(* POU TCP_Logger/LogEv, ST *)
FUNCTION LogEv : BOOL
VAR_INPUT
	Level	: en_Logger_ErrLev;
	Object  : en_SYS_Objects;
	Index	: WORD;
	Error	: WORD;
	Message : STRING;
END_VAR
VAR
	s1 : STRING(160);
	i  : INT;
END_VAR
(* Execute error level operations *)
CASE Level OF
	EL_Wrn: 		Sys.Warning:=TRUE;
	EL_Alarm: 		Sys.Alarm  :=TRUE;
	EL_AlarmStop: 	Sys.Alarm  :=TRUE; (* GO TO STOP STATE!! *)
END_CASE

(* Fill lastlog list *)
s1:=CONCAT(Sys.Time_LogString,';Lev=');
s1:=CONCAT(s1,INT_TO_STRING(Level));
s1:=CONCAT(s1,';Obj=');
s1:=CONCAT(s1,INT_TO_STRING(Object));
s1:=CONCAT(s1,';Idx=');
s1:=CONCAT(s1,WORD_TO_STRING(Index));
s1:=CONCAT(s1,';Err=');
s1:=CONCAT(s1,WORD_TO_STRING(Error));
Sys.LastLogs_Dat[Sys.LastLogs_Idx]:=s1;
Sys.LastLogs_Msg[Sys.LastLogs_Idx]:=Message;
Sys.LastLogs_Idx:=Sys.LastLogs_Idx+1;
IF Sys.LastLogs_Idx>5 THEN Sys.LastLogs_Idx:=0; END_IF

(*---------------------------------------------------------------*)
	Logger_Head();
(*---------------------------------------------------------------*)

(* Insert ERR *)
s1:=CONCAT('&ERR=',INT_TO_STRING(Level));
s1:=CONCAT(s1,';');
s1:=CONCAT(s1,INT_TO_STRING(Object));
s1:=CONCAT(s1,';');
s1:=CONCAT(s1,WORD_TO_STRING(Index));
s1:=CONCAT(s1,';');
s1:=CONCAT(s1,WORD_TO_STRING(Error));
s1:=CONCAT(s1,';');
ADDSTRING(ADR(Logger.TData), ADR(s1), Logger.TLen);
s1:=Message;
STR_NOSPACES(ADR(s1));
ADDSTRING(ADR(Logger.TData), ADR(s1), Logger.TLen);

(*---------------------------------------------------------------*)
	Logger_Send();
(*---------------------------------------------------------------*)
END_FUNCTION

(* POU Utils Functions/STR_NOSPACES, ST *)
FUNCTION STR_NOSPACES : BOOL (* Replace spaces and bad chars with allowed ones, used as HTTP-GET validator *)
VAR_INPUT
	pString: POINTER TO BYTE;
END_VAR
VAR
END_VAR
WHILE pString^<>0 DO
	IF pString^=16#20 (* space *) THEN pString^:=16#5F; (*'_'*) END_IF
	pString:=pString+1;
END_WHILE
END_FUNCTION

(* POU Utils Functions/AVERAGE_DINT, ST *)
FUNCTION_BLOCK AVERAGE_DINT
VAR_INPUT
	IN: 	DINT;
END_VAR
VAR_OUTPUT
	HI:		DINT;
	AVG:	DINT;
	LOW:	DINT;
	ERR:	BOOL;
END_VAR
VAR
	sum:	REAL;
	cnt:	WORD;
END_VAR
IF cnt>=65000 THEN
	ERR:=TRUE;
	Read();
	sum := sum - DINT_TO_REAL(AVG);
	cnt := cnt - 1;
END_IF

sum := sum + DINT_TO_REAL(IN);
cnt := cnt + 1;

IF IN<LOW THEN LOW:=IN; END_IF
IF IN>HI  THEN HI :=IN; END_IF
END_FUNCTION_BLOCK
ACTION Read:
AVG := REAL_TO_DINT(sum/cnt);
END_ACTION
ACTION Reset:
HI:=IN;
AVG:=IN;
LOW:=IN;
ERR:=FALSE;

sum:=DINT_TO_REAL(IN);
cnt:=1;
END_ACTION

(* POU Utils Functions/AVERAGE_INT, ST *)
FUNCTION_BLOCK AVERAGE_INT
VAR_INPUT
	IN: 	INT;
END_VAR
VAR_OUTPUT
	HI:		INT;
	AVG:	INT;
	LOW:	INT;
	ERR:	BOOL;
END_VAR
VAR
	sum:	DINT;
	cnt:	WORD;
END_VAR
IF cnt>=65000 THEN
	ERR:=TRUE;
	Read();
	sum := sum - AVG;
	cnt := cnt - 1;
END_IF

sum := sum + IN;
cnt := cnt + 1;

IF IN<LOW THEN LOW:=IN; END_IF
IF IN>HI  THEN HI :=IN; END_IF
END_FUNCTION_BLOCK
ACTION Read:
AVG := DINT_TO_INT(sum/cnt);
END_ACTION
ACTION Reset:
HI:=IN;
AVG:=IN;
LOW:=IN;
ERR:=FALSE;

sum:=IN;
cnt:=1;
END_ACTION

(* POU Utils Functions/AVERAGE_T, ST *)
FUNCTION_BLOCK AVERAGE_T
VAR_INPUT
	IN: 	INT;
END_VAR
VAR_OUTPUT
	HI:		INT;
	AVG:	INT;
	LOW:	INT;
	ERR:	BOOL;
END_VAR
VAR
	sum:	DINT;
	cnt:	WORD;
END_VAR
IF cnt>=65000 THEN
	ERR:=TRUE;
	Read();
	sum := sum - AVG;
	cnt := cnt + 1;
END_IF

sum := sum + IN;
cnt := cnt + 1;

IF IN<LOW THEN  LOW:=IN; END_IF
IF IN>HI  THEN HI :=IN; END_IF
END_FUNCTION_BLOCK
ACTION Read:
AVG := DINT_TO_INT(sum/cnt);
END_ACTION
ACTION Reset:
HI:=IN;
AVG:=IN;
LOW:=IN;
ERR:=FALSE;

sum:=IN;
cnt:=1;
END_ACTION

(* POU Utils Functions/BUILD_16TO32, ST *)
FUNCTION BUILD_16TO32 : DWORD
VAR_INPUT
		pSource	:	POINTER TO WORD;
END_VAR
VAR
		Data	:	DWORD;
END_VAR
Data := WORD_TO_DWORD(pSource^);
pSource := pSource + 1;
Data := Data + WORD_TO_DWORD(pSource^) * 65536;

BUILD_16TO32 := Data;
END_FUNCTION

(* POU Utils Functions/COPY_32SWAP16, ST *)
FUNCTION COPY_32SWAP16:BOOL
VAR_INPUT
	pSourceAddress		:POINTER TO ARRAY[1..2] OF WORD;
	pDestinationAddress	:POINTER TO ARRAY[1..2] OF WORD;
END_VAR
VAR
END_VAR
pDestinationAddress^[1]:=pSourceAddress^[2];
pDestinationAddress^[2]:=pSourceAddress^[1];
END_FUNCTION

(* POU Utils Functions/FLT_EVENT, ST *)
FUNCTION_BLOCK FLT_EVENT
VAR_INPUT
	IN		: BOOL;
	INITEV	: BOOL:=TRUE;
END_VAR
VAR_OUTPUT
	EVH		: BOOL;
	EVL		: BOOL;
END_VAR
VAR
	init	: BOOL:=FALSE;
	old		: BOOL;
END_VAR
EVH:=FALSE;
EVL:=FALSE;

IF NOT init THEN
	init:=TRUE;
	IF INITEV THEN
		old := NOT IN;
	ELSE
		old := IN;
	END_IF
END_IF

IF old<>IN THEN
	old:=IN;
	IF IN THEN EVH:=TRUE; ELSE EVL:=TRUE; END_IF
END_IF
END_FUNCTION_BLOCK

(* POU Utils Functions/FLT_TIME, ST *)
FUNCTION_BLOCK FLT_TIME
VAR_INPUT
	IN		: BOOL;
	TTAP	: TIME:=T#5s;
	INITEV	: BOOL:=TRUE;
END_VAR
VAR_OUTPUT
	OUT		: BOOL;
	EVH		: BOOL;
	EVL		: BOOL;
END_VAR
VAR
	init	: BOOL:=FALSE;
	timer	: TON;
END_VAR
EVH:=FALSE;
EVL:=FALSE;

IF NOT init THEN
	init := TRUE;
	IF INITEV THEN
		OUT  := NOT IN;
	ELSE
		OUT  := IN;
	END_IF
END_IF

IF OUT<>IN THEN
	timer(IN:=TRUE,PT:=TTAP);
	IF timer.Q THEN
		OUT:=IN;
		timer(IN:=FALSE);
		IF OUT THEN EVH:=TRUE; ELSE EVL:=TRUE; END_IF
	END_IF
ELSE
	timer(IN:=FALSE);
END_IF
END_FUNCTION_BLOCK

(* POU Utils Functions/LAMP_AL_GENERALE, ST *)
FUNCTION_BLOCK LAMP_AL_GENERALE
VAR_INPUT

	Allarme: BOOL;
	Warning: BOOL;
END_VAR
VAR_OUTPUT
	SistemaOK:BOOL;
	SistemaInAllarme:BOOL;
	SistemaWarning:BOOL;
	AllarmeLampada:BOOL;
END_VAR
VAR
	Lampeggio:BLINK;
END_VAR
IF Allarme THEN       					(* Se Allarme Attivo Lucde fissa ON *)
	SistemaInAllarme:=TRUE;
	SistemaWarning:=FALSE;
	AllarmeLampada:=TRUE;
ELSIF Warning THEN					(* Se Allarme Attivo Lucde fissa pulse *)
	SistemaInAllarme:=FALSE;
	SistemaWarning:=TRUE;
	Lampeggio(ENABLE:=TRUE , TIMELOW:=t#1s , TIMEHIGH:=t#1s , OUT=>AllarmeLampada );
ELSE
	SistemaInAllarme:=FALSE;
	SistemaWarning:=FALSE;
	AllarmeLampada:=FALSE;
END_IF
END_FUNCTION_BLOCK

(* POU Utils Functions/LINEAR, ST *)
FUNCTION LINEAR : REAL (* Linear interpolation *)
VAR_INPUT
	X_In	: REAL;
	P1_X	: REAL;
	P1_Y	: REAL;
	P2_X	: REAL;
	P2_Y	: REAL;
END_VAR
VAR
END_VAR
LINEAR:=P1_Y+(((P2_Y-P1_Y)*(X_In-P1_X))/(P2_X-P1_X));
END_FUNCTION

(* POU Utils Functions/LINEAR_BAD, ST *)
FUNCTION LINEAR_BAD : INT (* Linear interpolation *)
VAR_INPUT
	PuntoMinX	: INT;
	PuntoMaxX	: INT;
	ValIn		: INT;
	PuntoMinY	: REAL;
	PuntoMaxY	: REAL;
	Decimali	: BYTE;
END_VAR
VAR
	Gain				: REAL;
	PuntoMinX_R			: REAL;
	PuntoMaxX_R			: REAL;
	Linearizzazione_R	: REAL;
END_VAR
PuntoMinX_R:=INT_TO_REAL(PuntoMinX);
PuntoMaxX_R:=INT_TO_REAL(PuntoMaxX);

Gain:=(PuntoMaxX_R-PuntoMinX_R)/(PuntoMaxY-PuntoMinY);	(* Calcolo in guadagno per la linarizzazione *)
Linearizzazione_R:=PuntoMinx+(Gain*(ValIn-PuntoMinY));	(* Ottengo il valore linearizzato *)

LINEAR_BAD:=REAL_TO_INT(Linearizzazione_R*(EXPT(10, Decimali)));  (* Ottengo intero con i decimai voluti *)
END_FUNCTION

(* POU Utils Functions/MEAN_T, ST *)
FUNCTION MEAN_T : INT
VAR_INPUT
		T1		:	INT;
		T2		:	INT;

		THR_L	:	INT;
		THR_H	:	INT;
END_VAR
VAR
		Tmean	:	INT;
END_VAR
IF T1 >= THR_L AND T1 <= THR_H THEN

	IF T2 >= THR_L AND T2 <= THR_H THEN
		Tmean := (T1 + T2)/2;
	ELSE
		Tmean := T1;
	END_IF
ELSE
	IF T2 >= THR_L AND T2 <= THR_H THEN
		Tmean := T2;
	ELSE
		Tmean := 16#7FFF;	(* No valid temperature data has been passed *)
	END_IF
END_IF

MEAN_T := Tmean;
END_FUNCTION

(* POU Utils Functions/MEMCLR, ST *)
FUNCTION MEMCLR:BOOL
VAR_INPUT
	pDestinationAddress:POINTER TO ARRAY[1..2] OF BYTE;
	BytesToClear:WORD;
END_VAR
VAR
END_VAR
WHILE (BytesToClear > 0) DO
	pDestinationAddress^[1]:=0;
	pDestinationAddress:=ADR(pDestinationAddress^[2]); (* increment destination *)
	BytesToClear:=BytesToClear -1; (* decrement number of bytes to copy *)
END_WHILE
END_FUNCTION

(* POU Utils Functions/MUX_T, ST *)
FUNCTION MUX_T : INT
(* Manage temperatures measured by different probes in the same room/environment, considering possible probe measurement errors *)
VAR_INPUT
	T1		:	INT;
	T2		:	INT;
	T3		:	INT;
	(*T4		:	INT := 0;*)

	Err1	:	BOOL := TRUE;
	Err2	:	BOOL := TRUE;
	Err3	:	BOOL := TRUE;
	(*Err4	:	BOOL := TRUE;*)

	Used	:	BYTE;

END_VAR
VAR
	Sum		:	INT;
	count	:	BYTE;
END_VAR
CASE Used OF

	1:	(* T1 passed *)
		IF Err1 THEN
			Sum := 16#7FFF;
		ELSE
			Sum := T1;
			count := 1;
		END_IF

	2:	(* T1, T2 passed *)
		IF Err1 THEN
			IF Err2 THEN
				Sum := 16#7FFF;
			ELSE
				Sum := T2;
				count := 1;
			END_IF
		ELSE
			IF Err2 THEN
				Sum := T1;
				count := 1;
			ELSE
				Sum := T1 + T2;
				count := 2;
			END_IF
		END_IF

	3:	(* T1, T2, T3 passed *)
		IF Err1 THEN
			IF Err2 THEN
				IF Err3 THEN
					Sum := 16#7FFF;
				ELSE
					Sum := T3;
					count := 1;
				END_IF
			ELSE
				IF Err3 THEN
					Sum := T2;
					count := 1;
				ELSE
					Sum := T2 + T3;
					count := 2;
				END_IF
			END_IF
		ELSE
			IF Err2 THEN
				IF Err3 THEN
					Sum := T1;
					count := 1;
				ELSE
					Sum := T1 + T3;
					count := 2;
				END_IF
			ELSE
				IF Err3 THEN
					Sum := T1 + T2;
					count := 2;
				ELSE
					Sum := T1 + T2 + T3;
					count := 3;
				END_IF
			END_IF
		END_IF
(*
	4:
		IF Err1 THEN
			IF Err2 THEN
				IF Err3 THEN
					IF Err4 THEN
						Sum := 16#7FFF;
					ELSE
						Sum := T4;
						count := 1;
					END_IF
				ELSE
					IF Err4 THEN
						Sum := T3;
						count := 1;
					ELSE
						Sum := T3 + T4;
						count := 2;
					END_IF
				END_IF
			ELSE
				IF Err3 THEN
					IF Err4 THEN
						Sum := T2;
						count := 1;
					ELSE
						Sum := T2 + T4;
						count := 2;
					END_IF
				ELSE
					IF Err4 THEN
						Sum := T2 + T3;
						count := 2;
					ELSE
						Sum := T2 + T3 + T4;
						count := 3;
					END_IF
				END_IF
			END_IF
		ELSE
			IF Err2 THEN
				IF Err3 THEN
					IF Err4 THEN
						Sum := T1;
					ELSE
						Sum := T1 + T4;
						count := 2;
					END_IF
				ELSE
					IF Err4 THEN
						Sum := T1 + T3;
						count := 2;
					ELSE
						Sum := T1 + T3 + T4;
						count := 3;
					END_IF
				END_IF
			ELSE
				IF Err3 THEN
					IF Err4 THEN
						Sum := T1 + T2;
						count := 2;
					ELSE
						Sum := T1 + T2 + T4;
						count := 3;
					END_IF
				ELSE
					IF Err4 THEN
						Sum := T1 + T2 + T3;
						count := 3;
					ELSE
						Sum := T1 + T2 + T3 + T4;
						count := 4;
					END_IF
				END_IF
			END_IF
		END_IF
*)
END_CASE

IF Sum = 16#7FFF THEN
	(* No valid data -> return default *)
	MUX_T := Plant_DefaultTAmb;
ELSE
	(* Do average *)
	MUX_T := Sum/count;
END_IF
END_FUNCTION

(* POU Plant_Objects/obj_COOV_01, ST *)
FUNCTION_BLOCK obj_COOV_01
(* === ZIGBEE AMBIENT SENSORS MT-200 ===
   v1.0[07/05/05] - Create
*)
VAR CONSTANT
	LQI_Threshold		:	WORD := 10;		(* Zigbee link quality minimum value *)
	LowBattVoltage		:	WORD := 2700;		(* Battery is considered low when reaches 1.35V each *)
END_VAR
VAR_INPUT
	(* Settings *)
	ID				: BYTE;
	Address			: BYTE;

(*	Refresh_Period	: TIME:=t#5m;
	(* Controls *)
	Refresh_Auto	: BOOL:=TRUE; (* Enable automatic refresh *) *)
	(* Modbus *)
	Refresh_Now	:	BOOL;	(* Start immediately modbus state machine *)
	retryErrMax	:	BYTE := 2;


END_VAR
VAR_IN_OUT
	(* Interface *)
	ModBus		:obj_MODBUS;

END_VAR
VAR_OUTPUT
	(* Status *)
	Status_Log		: BYTE;
	Status_Vis 		: DWORD;
END_VAR
VAR


	state		:	INT;
	retry		:	BYTE;
	retryErr	:	BYTE;
	ReadTmr		:	TON := (PT:=T#5s);
	fModbusAlr:BOOL;


	AlarmCtr		: BYTE;
	WarningCtr		: BYTE;

	id_locale: BYTE;

	MB_RegistriLetti: ARRAY [0..20] OF INT;

	Quality			: FLT_EVENT;
	Battery			: FLT_EVENT;
	Alarm			: FLT_EVENT;

	ERR				: BOOL;
	fLQI			: BOOL;
	fBatt			: BOOL;
	StatusOK		: BYTE;			(* 0: Status OK, >=1: Alarm and/or warning		Incremented by 1 when Alarm or Wrn occurs,
									decremented by 1 when restored	*)

	TimeOutModBus: TON;
	ErroreComuModBus: BOOL;

	VerificaFuctionCode: INT;
	VerificaNodoLetto: INT;



END_VAR
(* stato creato per potere interrogare il nodo corretto *)
id_locale:=ID+6;

Stm();

checkAlarm();
END_FUNCTION_BLOCK
ACTION AddLogData:
Logger.s1:=INSERT('&COOV=',BYTE_TO_STRING(ID),5);
IF ID<10 THEN Logger.s1:=INSERT(Logger.s1,'0',5); END_IF


Logger.s1:=CONCAT(Logger.s1,INT_TO_STRING(MB_RegistriLetti[6]));	(* Misura del sensore CO2 – valore istantaneo  *)
Logger.s1:=CONCAT(Logger.s1,';');
Logger.s1:=CONCAT(Logger.s1,INT_TO_STRING(MB_RegistriLetti[4]));	(* Livello di Batteria (in millesimi di volt) *)
Logger.s1:=CONCAT(Logger.s1,';'); 
Logger.s1:=CONCAT(Logger.s1,WORD_TO_STRING(MB_RegistriLetti[3]));	(* Livello segnale radio dell'ultimo messaggio ricevuto dal dispositivo  *)
Logger.s1:=CONCAT(Logger.s1,';'); 

Logger.s1:=CONCAT(Logger.s1,BYTE_TO_STRING(Status_Log));
ADDSTRING(ADR(Logger.TData), ADR(Logger.s1), Logger.TLen);
END_ACTION
ACTION CheckAlarm:
(**** GEstione Log ad Evento *****)


(* (MB_RegistriLetti[3]) check Livello segnale radio dell'ultimo messaggio ricevuto dal dispositivo *)

IF (MB_RegistriLetti[3]) < LQI_Threshold THEN
	fLQI := FALSE;
	ERR := TRUE;
ELSE
	fLQI := TRUE;
	ERR := FALSE;
END_IF

Quality(IN:=fLQI);

IF Quality.EVL THEN
	LogEv(SEL((MB_RegistriLetti[3])<>0,EL_Alarm,EL_Wrn),EO_ZTHL,ID,SEL((MB_RegistriLetti[3])<>0,7,2),WORD_TO_STRING((MB_RegistriLetti[3])));
	Status_Log := SEL((MB_RegistriLetti[3])<>0,2,1);
	StatusOK := StatusOK + 1;
END_IF

IF Quality.EVH THEN StatusOK := SEL(StatusOK=0, StatusOK-1, 0); END_IF

(* If probe (node) is present proceed checking other warnings, otherwise don't transmit anything *)
IF (MB_RegistriLetti[3]) <> 0 THEN

	(* Check battery voltage *)

(* (MB_RegistriLetti[4]) check Livello di Batteria (in millesimi di volt) *)

	IF (MB_RegistriLetti[4]) < LowBattVoltage THEN fBatt := TRUE;
	ELSE fBatt := FALSE;
	END_IF


	Battery(IN:=fBatt);

	IF Battery.EVH  THEN
		LogEv(EL_Wrn,EO_ZTHL,ID,6,' ');
		StatusOK := StatusOK + 1;
	END_IF

	IF Battery.EVL THEN StatusOK := SEL(StatusOK=0, StatusOK-1, 0); END_IF

END_IF

Alarm(IN:=(StatusOK=0));

IF Alarm.EVH THEN
	Status_Log := 0;
	LogEv(EL_Log,EO_ZTHL,ID,1,'');
END_IF

IF Status_Log = 2 THEN Status_Vis := COLOR_RED;
ELSIF Status_Log = 1 THEN Status_Vis := COLOR_YELLOW;
ELSE Status_Vis := COLOR_GREEN;
END_IF
END_ACTION
ACTION Stm:
CASE state OF
	0:	(* Refresh time manager *)
		ReadTmr(IN:=NOT ReadTmr.Q);
		(*A tempo interrogo il nodo sempre che non ci sia qualcuno che lo sta interrogando in quel momento *)

		IF (ReadTmr.Q AND NodoDaInterrogareMB2=id_locale )OR Refresh_Now AND NOT InibiscoModbusMB2 THEN
			state := 10;
			ReadTmr.PT := T#5s;  (* moreno *)
			Refresh_Now := FALSE;
			InibiscoModbusMB2 := TRUE;
		END_IF

	(**** Leggo le Analogiche a Disposzione  ****)

	10:	(* richiedo lettura Holding Register   *)

		Modbus.MB_Query.SlaveAddress := Address;
		Modbus.MB_Query.FunctionCode := 4;
		ModBus.MB_Query.Read_StartAddress := 0 ;			(* richiedo lettura altri Parametri *)
		ModBus.MB_Query.Read_Quantity := 8;
		ModBus.MB_Start := TRUE;
		state := 20;

	20:	(* Risposta all'interrogazione *)
		IF NOT ModBus.MB_Start   THEN
			VerificaFuctionCode:=ModBus.MB_Resp.FunctionCode;
			VerificaNodoLetto:=ModBus.MB_Resp.SlaveAddress;

			IF ModBus.MB_MASTER.MB_Error<>0 THEN
				state := 300;
			ELSE

				MB_RegistriLetti[0] := ModBus.MB_Resp.Data[0];   	(* Vedi tabella *)
				MB_RegistriLetti[1] := ModBus.MB_Resp.Data[1];		(* Vedi tabella *)
				MB_RegistriLetti[2] := ModBus.MB_Resp.Data[2];		(* Vedi tabella *)
				MB_RegistriLetti[3] := ModBus.MB_Resp.Data[3];		(* Vedi tabella *)
				MB_RegistriLetti[4] := ModBus.MB_Resp.Data[4];		(* Vedi tabella *)
				MB_RegistriLetti[5] := ModBus.MB_Resp.Data[5];		(* Vedi tabella *)
				MB_RegistriLetti[6] := ModBus.MB_Resp.Data[6];		(* Vedi tabella *)
				MB_RegistriLetti[7] := ModBus.MB_Resp.Data[7];		(* Vedi tabella *)
				MB_RegistriLetti[8] := ModBus.MB_Resp.Data[8];		(* Vedi tabella *)
				MB_RegistriLetti[9] := ModBus.MB_Resp.Data[9];		(* Vedi tabella *)
				MB_RegistriLetti[10] := ModBus.MB_Resp.Data[10];		(* Vedi tabella *)
				MB_RegistriLetti[11] := ModBus.MB_Resp.Data[11];		(* Vedi tabella *)
				MB_RegistriLetti[12] := ModBus.MB_Resp.Data[12];		(* Vedi tabella *)
				MB_RegistriLetti[13] := ModBus.MB_Resp.Data[13];		(* Vedi tabella *)

				state := 295;
			END_IF
		END_IF


		295:
		IF NOT ModBus.MB_Start THEN
			IF ModBus.MB_MASTER.MB_Error<>0 THEN (*OR ModBus.MB_MASTER.MB_Error<>0 THEN*)
				state := 300;
			ELSE
				IF fModbusAlr THEN fModbusAlr := FALSE; END_IF
				NodoDaInterrogareMB2:=id_locale+1;
				InibiscoModbusMB2:=FALSE;
				retryErr := 0;
				retry := 0;
				state := 0;
					IF fModbusAlr=FALSE AND ErroreComuModBus=TRUE THEN
						LogEv(EL_Log,EO_CHI,ID,62,'ComunicazioneModBus_OK');
						ErroreComuModBus := FALSE;
				(*	WarningCtr := SEL(WarningCtr=0, WarningCtr-1, 0); *)
					END_IF


			END_IF
		END_IF



	(**** CHECK MODBUS ERROR ****)
	300: 	(* Release MODBUS *)
			InibiscoModbusMB2:=FALSE;
			(* Retries *)
			retry:=retry+1;
			IF retry>3 THEN
				retry:=0;

				(* Verify if slave is dead *)
				IF retryErr < retryErrMaX THEN
					retryErr := retryErr + 1;
				ELSE
					fModbusAlr := TRUE;
					(* Verify ModBus error	*)

					IF fModbusAlr AND ErroreComuModBus=FALSE THEN
						LogEv(EL_Alarm,EO_CHI,ID,61,CONCAT('ErroreModbus_',INT_TO_STRING(ModBus.MB_MASTER.MB_Error)));
						ErroreComuModBus := TRUE;
					END_IF
				END_IF

				END_IF
			Refresh_Now := FALSE;
			InibiscoModbusMB2:=FALSE;
			NodoDaInterrogareMB2:=id_locale+1;
			state:=0;
END_CASE




(* Controllo Time Out Ciclo ModBus *)

TimeOutModBus(In:=state<>0,PT:=t#30s);
IF TimeOutModBus.Q THEN
	State:=0;
	Refresh_Now:=TRUE;  (* Rilancio la lettura del nodo *)
	IF MODBUS.MB_Lock=TRUE THEN MODBUS.MB_Lock:=FALSE;END_IF
	IF InibiscoModbusMB2=TRUE THEN InibiscoModbusMB2:=FALSE;END_IF
END_IF
END_ACTION

(* POU Plant_Objects/obj_MODBUS, ST *)
FUNCTION_BLOCK obj_MODBUS
(* === MODBUS PROTOCOL INTERFACE ===
   v1.1[19/06/15] - Added new VARS allocation and searching
*)
VAR CONSTANT
	VARS_Max	: BYTE := 32;
END_VAR
VAR_INPUT
	(* Settings *)
	ID			: BYTE;
	COM			: BYTE;
	BAUDRATE	: COM_BAUDRATE;
	RS485		: BOOL := FALSE;

	N_STOPBits	:BYTE:=1;

	(* Interface *)
	MB_MASTER	: MODBUS_EXTENDED_MASTER;
	MB_Start	: BOOL;
	MB_Query	: typModbusExtendedQuery;
	MB_Resp		: typModbusResponse;
	MB_Lock		: BOOL;
	MB_timeOut	: TIME := t#500ms;

	(* Variables management *)
	VARS_En		: BOOL;
	VARS		: ARRAY [0..VARS_Max] OF typ_MODBUS_VAR;
	VARS_Check	: BOOL;
	VARS_Alarm	: BOOL;

	(* Variables allocation *)
	VAR_Pointer : POINTER TO ARRAY[0..99] OF WORD;
	VAR_Cfg		: POINTER TO typ_MODBUS_VAR;
END_VAR
VAR_OUTPUT
	(* Status *)
	Status_Log	: BYTE;
	Status_Vis	: DWORD;
END_VAR
VAR
	sta         : BYTE :=0;
	i			: BYTE;
	j			: BYTE;
	Alarm		: FLT_EVENT;
	
	VarTmr		: TON := (PT:=T#1s);
	VarSta		: BYTE; (* Status *)
	VarCnt		: BYTE; (* Scan counter *)
	VarRetry	: BYTE;
	VarAlarm	: BYTE; (* Last variable with errors *)
END_VAR
IF N_STOPBits=1 THEN MB_MASTER.csCOM_STOPBITS:=STOPBITS_1;END_IF
IF N_STOPBits=2 THEN MB_MASTER.csCOM_STOPBITS:=STOPBITS_2;END_IF

MB_MASTER(ENABLE:=TRUE,	ASCII_Mode:=FALSE, bCOM_PORT:=COM, cbCOM_BAUDRATE:=BAUDRATE, cpCOM_PARITY:=PARITY_NO,
		cbsCOM_BYTESIZE:=BS_8, cfCOM_FLOW_CONTROL:=SEL(RS485,NO_FLOW_CONTROL,HALFDUPLEX),
		tTIME_OUT:=MB_timeOut,	StartFunction:=MB_Start, ExtQuery:=MB_Query, Response:=MB_Resp);

(* Process variable management *)
IF VARS_En THEN VARS_Process(); END_IF

(* Check status *)
Alarm(IN:=(MB_MASTER.bInterfaceError<>0));
IF Alarm.EVH THEN
	LogEv(SEL(MB_MASTER.bInterfaceError<>3,EL_Wrn,EL_Alarm),EO_MODBUS,ID,1,BYTE_TO_STRING(MB_MASTER.bInterfaceError));
END_IF
IF Alarm.EVL THEN								(* Trigger a fall edge: MODBUS back working *)
	LogEv(EL_Log,EO_MODBUS,ID,2,'MODBUS_OK');
END_IF

(* Log/visu status *)
   IF Alarm.IN   THEN Status_Log:=2; Status_Vis:=COLOR_RED;
ELSIF Vars_Alarm THEN Status_Log:=1; Status_Vis:=COLOR_YELLOW;
  				 ELSE Status_Log:=0; Status_Vis:=COLOR_GREEN;
END_IF
END_FUNCTION_BLOCK
ACTION VAR_Search:
(* Search VAR with specific pointer if not found return first free VAR
	[Last VAR is not active... used as safe area...] 
*)
j:=VARS_Max;
FOR i := 0 TO VARS_Max-1 DO
	IF VARS[i].Variable=0 AND j>i THEN j:=i; END_IF
	IF VARS[i].Variable=VAR_Pointer THEN
		VAR_Cfg:=ADR(VARS[i]);
		RETURN;
	END_IF
END_FOR
VAR_Cfg:=ADR(VARS[j]);
END_ACTION
ACTION VARS_Process:
(* Update var timers *)
VarTmr(IN:=(NOT VarTmr.Q));
IF VarTmr.Q THEN
	FOR i := 0 TO VARS_Max DO
		IF VARS[i].Refresh_Cnt>0 THEN VARS[i].Refresh_Cnt:=VARS[i].Refresh_Cnt-1; END_IF
	END_FOR
	VARS_Check:=TRUE;
END_IF


(* Process status *)
CASE VarSta OF
	0: (* === Init *)
		VarCnt:=0;
		VarSta:=1;

	1: (* === Wait check signal *)
		IF VARS_Check THEN				(* Decremented "Refresh_Cnt" *)
			VARS_Check:=FALSE;
			VarCnt:=0;
			VarSta:=2;
		END_IF

	2: (* === Check loop *)
		IF NOT (MB_Lock OR MB_Start) THEN
			WHILE VarCnt<=(VARS_Max-1) AND VarSta=2 DO
				(* Check only active vars *)
				IF VARS[VarCnt].Variable<>0 THEN			(* "Variable" is a pointer to word, so if 0 no address *)
					(* Check var auto-refresh on timer checks *)
					IF VARS[VarCnt].Refresh_Time>0 AND VARS[VarCnt].Refresh_Cnt=0 THEN
						VARS[VarCnt].Refresh_Cnt:=VARS[VarCnt].Refresh_Time;
						VarSta:=3;
					END_IF
					(* Check refresh for change or request *)
					CASE VARS[VarCnt].FunCode OF
						5,6,15,16: (* Write functions *)
							IF VARS[VarCnt].Variable_Size=1 THEN
								IF VARS[VarCnt].Variable^<>VARS[VarCnt].Variable_Mirror THEN
									VARS[VarCnt].Variable_Mirror:=VARS[VarCnt].Variable^;
									VarSta:=3;
								END_IF
							ELSE
								IF VARS[VarCnt].Variable_Mirror<>0 THEN
									VARS[VarCnt].Variable_Mirror:=0;
									VarSta:=3;
								END_IF
							END_IF
						1,2,3,4: (* Read functions *)
							IF VARS[VarCnt].Variable_Mirror<>0 THEN
								VARS[VarCnt].Variable_Mirror:=0;
								VarSta:=3;
							END_IF
					END_CASE
				END_IF
				(* Process query *)
				IF VarSta=3 THEN
					MB_Lock:=TRUE;
					MB_Query.SlaveAddress:=VARS[VarCnt].SlaveAddress;
					MB_Query.FunctionCode:=VARS[VarCnt].FunCode;
					CASE VARS[VarCnt].FunCode OF
						16#5,16#6,16#F,16#10:
							MB_Query.Read_Quantity:=0;
							MB_Query.Read_StartAddress:=0;
							MB_Query.Write_StartAddress:=VARS[VarCnt].FunAddress;
							MB_Query.Write_Quantity:=VARS[VarCnt].Variable_Size;
							IF VARS[VarCnt].Variable_Size=200 THEN
								COPY_32SWAP16(VARS[VarCnt].Variable, ADR(MB_Query.Write_Data[0]));
							ELSIF VARS[VarCnt].Variable_Size>1 THEN
								MEMCPY(VARS[VarCnt].Variable, ADR(MB_Query.Write_Data[0]), 2*VARS[VarCnt].Variable_Size);
							ELSE
								MB_Query.Write_Data[0]:=VARS[VarCnt].Variable^;
							END_IF
						16#1,16#2,16#3,16#4:
							MB_Query.Read_StartAddress:=VARS[VarCnt].FunAddress;
							IF VARS[VarCnt].Variable_Size=200 THEN MB_Query.Read_Quantity:=2; ELSE
							  MB_Query.Read_Quantity:=VARS[VarCnt].Variable_Size;
							END_IF
							MB_Query.Write_StartAddress:=0;
							MB_Query.Write_Quantity:=0;
					END_CASE
					VarRetry:=0;
					MB_Start:=TRUE;
				ELSE
					VarCnt:=VarCnt+1;
				END_IF
			END_WHILE
			(* Check loop completed -> no actions *)
			IF VarSta=2 THEN VarSta:=1; END_IF
		END_IF

	3: (* === Wait & process MB response *)
		IF NOT MB_Start THEN
			IF MB_MASTER.MB_Error=0 THEN
				CASE VARS[VarCnt].FunCode OF
					1,2,3,4:
						IF VARS[VarCnt].Variable_Size=200 THEN
							COPY_32SWAP16(ADR(MB_Resp.Data), VARS[VarCnt].Variable);
						ELSIF VARS[VarCnt].Variable_Size>1 THEN
							MEMCPY(ADR(MB_Resp.Data), VARS[VarCnt].Variable, 2*VARS[VarCnt].Variable_Size);
						ELSE
							VARS[VarCnt].Variable^:=MB_Resp.Data[0];
						END_IF
				END_CASE
				MB_Lock:=FALSE;
				(* Signal error recovery *)
				IF VARS_Alarm=TRUE AND VarCnt=VarAlarm THEN
					LogEv(EL_Wrn,EO_MODBUS,ID,5,'');
					VARS_Alarm:=FALSE;
				END_IF
				(* Next var *)
				VarCnt:=VarCnt+1;
				VarSta:=2;
			ELSE
				IF VarRetry<3 THEN
					VarRetry:=VarRetry+1;
					MB_Start:=TRUE;
				ELSE
					MB_Lock:=FALSE;
					(* Signal error *)
					IF VARS_Alarm=FALSE THEN
						LogEv(EL_Wrn,EO_MODBUS,ID,3,INT_TO_STRING(MB_MASTER.MB_Error));
						VARS_Alarm:=TRUE;
						VarAlarm:=VarCnt-1;
					END_IF
					(* Next var *)
					VarCnt:=VarCnt+1;
					VarSta:=2;
				END_IF
			END_IF
		END_IF

ELSE
	VarSta:=0;
END_CASE
END_ACTION

(* POU Plant_Objects/obj_CRON, ST *)
FUNCTION_BLOCK obj_CRON
(* === CRONOGRAFO STANDARD ===
   v1.0[16/04/15] - Versioning
   v1.1[19/05/15] - Removed DB creation from previous year
*)
VAR_INPUT
	(* Settings *)
	ID			: BYTE;		(* Index of instanced object *)

	InitOK		: BOOL;
	Alarm		: BOOL;
	Warning		: BOOL;

	Profile		: typ_Cron_Profile; 				(* Profilo attivo *)
	ProfileNr	: BYTE;								(* Indice profilo attivo *)
	CalendarIdx : WORD;								(* Indice calendario attivo *)
	Jolly		: ARRAY[0..9] OF typ_Cron_Jolly;	(* Jolly attivi *)

END_VAR
VAR_IN_OUT
END_VAR
VAR_OUTPUT
	SetPoint		: INT;
	(* Status *)
	Status_Log		: BYTE;
	Status_Vis 		: DWORD;
END_VAR
VAR
	Buf: 	ARRAY[0..512] OF BYTE; (* AVOID THIS!! *)
	hFile: 	DWORD;
	sFile: 	STRING;
	sFile2: STRING;

	i:		WORD;
	t1:		DWORD;
	t2:		BOOL;

END_VAR
(* Check initialization *)
IF NOT InitOK THEN Init(); END_IF

(* Chrono *)
IF CalendarIdx<>Sys.Time_CT_Day THEN DB_Load(); END_IF
SetPoint:=Profile.Setpoint[Sys.Time_CT_Quarter];

(* Check jolly *)
FOR i := 0 TO 9 DO
	IF ( DT_TO_DWORD(Jolly[i].Start)>0  AND Jolly[i].End>Jolly[i].Start AND
	     Jolly[i].Start<=Sys.Time_CT_DT AND Jolly[i].End>Sys.Time_CT_DT ) THEN
			SetPoint:=Jolly[i].Temp;
	END_IF
END_FOR


(* Status color *)
   IF Alarm   THEN Status_Log:=2; Status_Vis:=COLOR_RED;
ELSIF Warning THEN Status_Log:=1; Status_Vis:=COLOR_YELLOW;
              ELSE Status_Log:=0; Status_Vis:=COLOR_GREEN;
			  END_IF
END_FUNCTION_BLOCK
ACTION AddLogData:
Logger.s1:=INSERT('&CRON=',BYTE_TO_STRING(ID),5);
IF ID<10 THEN Logger.s1:=INSERT(Logger.s1,'0',5); END_IF

Logger.s1:=CONCAT(Logger.s1,INT_TO_STRING(SetPoint));			Logger.s1:=CONCAT(Logger.s1,';');

Logger.s1:=CONCAT(Logger.s1,WORD_TO_STRING(Status_Log));
ADDSTRING(ADR(Logger.TData), ADR(Logger.s1), Logger.TLen);
END_ACTION
ACTION DB_Create:
(* Create empty file *)
hFile:=SysFileOpen(FileName:=sFile, Mode:='w');

MEMCLR(pDestinationAddress:=ADR(Buf), BytesToClear:=SIZEOF(Buf));
FOR i := 0 TO 10239 BY 512 DO
	t1:=SysFileWrite(File:=hFile, Buffer:=ADR(Buf), Size:=512);		(* Clear created file (all bytes 0) *)
END_FOR
Buf[0]:=1;
t2:=SysFileSetPos(File:=hFile, Pos:=0);
t1:=SysFileWrite(File:=hFile, Buffer:=ADR(Buf), Size:=1);
SysFileClose(File:=hFile);
END_ACTION
ACTION DB_Load:
DB_SetName();

(* Open data file *)
hFile:=SysFileOpen(FileName:=sFile, Mode:='r');

(* File not found *)
IF hFile=0 THEN
	Warning:=TRUE;
	LogEv(EL_Wrn,EO_CRON,ID,1,'No_data_file');
	DB_Create();
	(* Reopen file *)
	hFile:=SysFileOpen(FileName:=sFile, Mode:='r');
	IF hfile=0 THEN
		Alarm:=TRUE;
		LogEv(EL_Alarm,EO_CRON,ID,3,'Filesystem_error');
		RETURN;
	END_IF
END_IF

(* Check version *)
SysFileRead(File:=hFile, Buffer:=ADR(Buf), Size:=1);
IF Buf[0]<>1 THEN
	IF NOT Alarm THEN
		Alarm:=TRUE;
		LogEv(EL_Alarm,EO_CRON,ID,2,'Bad_data_version');
	END_IF
	SysFileClose(File:=hFile);
	RETURN;
END_IF

(* Read Jolly data *)
t2:=SysFileSetPos(File:=hFile, Pos:=512);
t1:=SysFileRead(File:=hFile, Buffer:=ADR(Jolly), Size:=SIZEOF(Jolly));
(* Read active profile index *)
CalendarIdx:=Sys.Time_CT_Day;
t2:=SysFileSetPos(File:=hFile, Pos:=(1024+4*CalendarIdx));
t1:=SysFileRead(File:=hFile, Buffer:=ADR(ProfileNr), Size:=SIZEOF(ProfileNr));
(* Read active profile *)
t2:=SysFileSetPos(File:=hFile, Pos:=(3072+512*ProfileNr));
t1:=SysFileRead(File:=hFile, Buffer:=ADR(Profile), Size:=SIZEOF(Profile));

(* Close file and validate data *)
SysFileClose(File:=hFile);
END_ACTION
ACTION DB_SetName:
(* Create current filename 'yyyyCRnn.DAT' *)
sFile:=CONCAT(FilesPath,WORD_TO_STRING(Sys.Time_Year));
sFile:=CONCAT(STR1:=sFile, STR2:='CR');
IF ID<10 THEN
sFile:=CONCAT(STR1:=sFile, STR2:='0');
END_IF
sFile:=CONCAT(STR1:=sFile, STR2:=BYTE_TO_STRING(ID));
sFile:=CONCAT(STR1:=sFile, STR2:='.DAT');
END_ACTION
ACTION Init:
DB_Load();
InitOK:=TRUE;
END_ACTION

(* POU Plant_Objects/obj_CRON_EDITOR, ST *)
FUNCTION_BLOCK obj_CRON_EDITOR
(* === EDITOR CRONOGRAFO ===
   v1.0[16/04/15] - Versioning
   v1.1[19/05/15] - Create empty profile when not found
*)
VAR_INPUT

	(* Common selections *)
	CN_Sel:			BYTE:=1;
	CN_Act:			BYTE;
	CN_YSel:		WORD:=2015;
	CN_YAct:		WORD;

	(* Profile editor *)
	PR_Sel: 		BYTE:=1;
	PR_Act:			BYTE;
	PR_TT:			REAL;
	PR:				typ_Cron_Profile;
	(* Profile signals *)
	PR_Load:		BOOL;
	PR_Save:		BOOL;

	(* Calendar editor *)
	CA_Sel:			BYTE:=1; (* Calendar month selected *)
	CA_Act:			BYTE;    (* Calendar month active *)
	CA_DayF:		BYTE:=0;
	CA_DayL:		BYTE:=31;
	CA_TPR:			BYTE;
	CA:				typ_Cron_Calendar; (* Only used for first 32 entries *)
	(* Calendar signals *)
	CA_Load:		BOOL;
	CA_Save:		BOOL;

	(* Jolly editor *)
	JL:				ARRAY[0..9] OF typ_Cron_Jolly;
	(* Jolly signals *)
	JL_Load:		BOOL;
	JL_Save:		BOOL;

END_VAR
VAR_OUTPUT
	Message		: STRING;
END_VAR
VAR
	sFileName	: STRING;
	sFileMode	: STRING;
	hFile		: DWORD;
	Buf			: ARRAY[0..512] OF BYTE; (* AVOID THIS!! *)

	i			: WORD;
	ver			: BYTE;
	r1			: BOOL;
	r2			: DWORD;

END_VAR
IF PR_Load THEN PR_Load_Exe(); PR_Load:=FALSE; END_IF
IF PR_Save THEN PR_Save_Exe(); PR_Save:=FALSE; END_IF
IF CA_Load THEN CA_Load_Exe(); CA_Load:=FALSE; END_IF
IF CA_Save THEN CA_Save_Exe(); CA_Save:=FALSE; END_IF
IF JL_Load THEN JL_Load_Exe(); JL_Load:=FALSE; END_IF
IF JL_Save THEN JL_Save_Exe(); JL_Save:=FALSE; END_IF
END_FUNCTION_BLOCK
ACTION CA_Load_Exe:
sFileMode:='r';
FileOpen();

IF hFile<>0 THEN

	(* Read calendar month *)
	FOR i := 0 TO 31 DO
		r1:=SysFileSetPos(File:=hFile, Pos:=(1024 + ((CA_Sel-1)*32 + i)*4));
		r2:=SysFileRead(File:=hFile, Buffer:=ADR(CA.Profile[i]), Size:=1);
	END_FOR

	(* Close file *)
	SysFileClose(File:=hFile);

	(* Validate data *)
	CA_Act :=CA_Sel;
	CN_Act :=CN_Sel;
	CN_YAct:=CN_YSel;

	Message:='Calendar load OK';

END_IF
END_ACTION
ACTION CA_Save_Exe:
sFileMode:='a';
FileOpen();

IF hFile<>0 THEN

	(* Write calendar month *)
	FOR i := 0 TO 31 DO
		r1:=SysFileSetPos(File:=hFile, Pos:=(1024 + ((CA_Sel-1)*32 + i)*4));
		r2:=SysFileGetPos(hFile);
		r2:=SysFileWrite(File:=hFile, Buffer:=ADR(CA.Profile[i]), Size:=1);
	END_FOR

	(* Close file *)
	SysFileClose(File:=hFile);

	Message:='Calendar save OK';

END_IF
END_ACTION
ACTION FileOpen:
(* Create current filename 'yyyyCRnn.DAT' *)
sFileName:=CONCAT(FilesPath,WORD_TO_STRING(CN_YSel));
sFileName:=CONCAT(STR1:=sFileName, STR2:='CR');
IF CN_Sel<10 THEN
sFileName:=CONCAT(STR1:=sFileName, STR2:='0');
END_IF
sFileName:=CONCAT(STR1:=sFileName, STR2:=BYTE_TO_STRING(CN_Sel));
sFileName:=CONCAT(STR1:=sFileName, STR2:='.DAT');

(* Check file version and size! *)
(* ... *)

(* Open data file *)
hFile:=SysFileOpen(FileName:=sFileName, Mode:='r');

(* File not found *)
IF hFile=0 THEN
	Message:='File not found - created empty file';
	(* Create empty file *)
	hFile:=SysFileOpen(FileName:=sFileName, Mode:='w');
	MEMCLR(pDestinationAddress:=ADR(Buf), BytesToClear:=SIZEOF(Buf));
	FOR i := 0 TO 10239 BY 512 DO
		SysFileWrite(File:=hFile, Buffer:=ADR(Buf), Size:=512);
	END_FOR
	Buf[0]:=1;
	SysFileSetPos(File:=hFile, Pos:=0);
	SysFileWrite(File:=hFile, Buffer:=ADR(Buf), Size:=1);
END_IF

(* Close file *)
SysFileClose(File:=hFile);

(* Open data file *)
hFile:=SysFileOpen(FileName:=sFileName, Mode:=sFileMode);
END_ACTION
ACTION JL_Load_Exe:
sFileMode:='r';
FileOpen();

IF hFile<>0 THEN

	(* Read jolly *)
	r1:=SysFileSetPos(File:=hFile, Pos:=512);
	r2:=SysFileRead(File:=hFile, Buffer:=ADR(JL), Size:=SIZEOF(JL));

	(* Close file *)
	SysFileClose(File:=hFile);

	(* Validate data *)
	CN_Act:=CN_Sel;
	CN_YAct:=CN_YSel;

	Message:='Jolly load OK';

END_IF
END_ACTION
ACTION JL_Save_Exe:
sFileMode:='a';
FileOpen();

IF hFile<>0 THEN

	(* Write selected profile *)
	r1:=SysFileSetPos(File:=hFile, Pos:=512);
	r2:=SysFileWrite(File:=hFile, Buffer:=ADR(JL), Size:=SIZEOF(JL));

	(* Close file *)
	SysFileClose(File:=hFile);

	Message:='Jolly save OK';

END_IF
END_ACTION
ACTION PR_Load_Exe:
sFileMode:='r';
FileOpen();

IF hFile<>0 THEN

	(* Read selected profile *)
	r1:=SysFileSetPos(File:=hFile, Pos:=(3072 + 512*PR_Sel));
	r2:=SysFileRead(File:=hFile, Buffer:=ADR(PR), Size:=SIZEOF(PR));

	(* Close file *)
	SysFileClose(File:=hFile);

	(* Validate data *)
	PR_Act:=PR_Sel;
	CN_Act:=CN_Sel;
	CN_YAct:=CN_YSel;

	Message:='Profile load OK';

END_IF
END_ACTION
ACTION PR_Save_Exe:
sFileMode:='a';
FileOpen();

IF hFile<>0 THEN

	(* Write selected profile *)
	r1:=SysFileSetPos(File:=hFile, Pos:=(3072 + 512*PR_Sel));
	r2:=SysFileWrite(File:=hFile, Buffer:=ADR(PR), Size:=SIZEOF(PR));

	(* Close file *)
	SysFileClose(File:=hFile);

	Message:='Profile save OK';

END_IF
END_ACTION

(* POU Plant_Objects/obj_CRONTER, ST *)
FUNCTION_BLOCK obj_CRONTER
(* === THERMOSTAT ===
   v1.0[30/07/15] - Versioning
*)
VAR_INPUT
	(* Settings *)
	ID			: BYTE;		(* Index of instanced object *)

	InitOK		: BOOL;
	Alarm		: BOOL;
	Warning		: BOOL;

	Profile		: typ_Cron_Profile; 				(* Profilo attivo *)
	ProfileNr	: BYTE;								(* Indice profilo attivo *)
	CalendarIdx : WORD;								(* Indice calendario attivo *)
	Jolly		: ARRAY[0..9] OF typ_Cron_Jolly;	(* Jolly attivi *)

	Temperature	: INT;
	Local_MaxRunTAmb	:	INT;					(* Local maximum environment temperature, NOT "TAMB" *)

	Histeresys:INT; (* isteresi per la ripartenza del Comando ON*)
END_VAR
VAR_IN_OUT
END_VAR
VAR_OUTPUT
	SetPoint		: INT;
	Run				: BOOL;
	AntifreezeForce	: BOOL;
	RunCrono		: BOOL;

	(* Status *)
	Status_Log		: BYTE;
	Status_Vis 		: DWORD;
END_VAR
VAR
	Buf: 	ARRAY[0..512] OF BYTE; (* AVOID THIS!! *)
	hFile: 	DWORD;
	sFile: 	STRING;
	sFile2: STRING;

	i:		WORD;
	t1:		DWORD;
	t2:		BOOL;

END_VAR
(* Check initialization *)
IF NOT InitOK THEN Init(); END_IF

(* Check Temperature *)
(*IF Temperature < Local_MaxRunTAmb THEN*)

	(* LOCAL environment temperature lower than maximum allowed -> Proceed with SetPoint adjustment *)
	(* Chrono *)
	IF CalendarIdx<>Sys.Time_CT_Day THEN DB_Load(); END_IF
	SetPoint:=Profile.Setpoint[Sys.Time_CT_Quarter];

	(* Check jolly *)
	FOR i := 0 TO 9 DO
		IF ( DT_TO_DWORD(Jolly[i].Start)>0  AND Jolly[i].End>Jolly[i].Start AND
		     Jolly[i].Start<=Sys.Time_CT_DT AND Jolly[i].End>Sys.Time_CT_DT ) THEN
				SetPoint:=Jolly[i].Temp;
		END_IF
	END_FOR

(*
	IF SetPoint < 180 THEN
		(* Switch off the device *)
		Run := FALSE;
	ELSE
		(* Set according to feedback T - Histeresys of 1°C *)
		IF Temperature >= (SetPoint + 5) THEN
			Run := FALSE;
		ELSIF Temperature <= (SetPoint - 5) THEN
			Run := TRUE;
		END_IF

		(* Between "SetPoint-5" and "SetPoint+5" last state (ON or OFF) of "Run" is kept	*)
	END_IF
*)

(* Gestione uscita Crono *)
		IF SetPoint>0 THEN RunCrono := TRUE;
		ELSIF SetPoint=0 THEN RunCrono := FALSE;
		END_IF

(* GEstione uscita Cronotermostato *)


		IF Temperature >= (SetPoint) THEN
			Run := FALSE;
		ELSIF Temperature <= (SetPoint - Histeresys) THEN
			Run := TRUE;
		END_IF


(*ELSE
	(* Environment overtemperature: stop heating -> Stop device *)
	Run := FALSE;
END_IF
*)
(* Freeze warning: Switch on and heat! *)
(*IF Temperature < Plant_AntiFreezeTAmb THEN AntifreezeForce := TRUE;
ELSE AntifreezeForce := FALSE;
END_IF*)



(* Status color *)
   IF Alarm   THEN Status_Log:=2; Status_Vis:=COLOR_RED;
ELSIF Warning THEN Status_Log:=1; Status_Vis:=COLOR_YELLOW;
              ELSE Status_Log:=0; Status_Vis:=COLOR_GREEN;
			  END_IF
END_FUNCTION_BLOCK
ACTION AddLogData:
Logger.s1:=INSERT('&THER=',BYTE_TO_STRING(ID),5);
IF ID<10 THEN Logger.s1:=INSERT(Logger.s1,'0',5); END_IF

Logger.s1:=CONCAT(Logger.s1,INT_TO_STRING(SetPoint));			Logger.s1:=CONCAT(Logger.s1,';');

Logger.s1:=CONCAT(Logger.s1,WORD_TO_STRING(Status_Log));
ADDSTRING(ADR(Logger.TData), ADR(Logger.s1), Logger.TLen);
END_ACTION
ACTION DB_Create:
(* Create empty file *)
hFile:=SysFileOpen(FileName:=sFile, Mode:='w');

MEMCLR(pDestinationAddress:=ADR(Buf), BytesToClear:=SIZEOF(Buf));
FOR i := 0 TO 10239 BY 512 DO
	t1:=SysFileWrite(File:=hFile, Buffer:=ADR(Buf), Size:=512);		(* Clear created file (all bytes 0) *)
END_FOR
Buf[0]:=1;
t2:=SysFileSetPos(File:=hFile, Pos:=0);
t1:=SysFileWrite(File:=hFile, Buffer:=ADR(Buf), Size:=1);
SysFileClose(File:=hFile);
END_ACTION
ACTION DB_Load:
DB_SetName();

(* Open data file *)
hFile:=SysFileOpen(FileName:=sFile, Mode:='r');

(* File not found *)
IF hFile=0 THEN
	Warning:=TRUE;
	LogEv(EL_Wrn,EO_CRON,ID,1,'No_data_file');
	DB_Create();
	(* Reopen file *)
	hFile:=SysFileOpen(FileName:=sFile, Mode:='r');
	IF hfile=0 THEN
		Alarm:=TRUE;
		LogEv(EL_Alarm,EO_CRON,ID,3,'Filesystem_error');
		RETURN;
	END_IF
END_IF

(* Check version *)
SysFileRead(File:=hFile, Buffer:=ADR(Buf), Size:=1);
IF Buf[0]<>1 THEN
	IF NOT Alarm THEN
		Alarm:=TRUE;
		LogEv(EL_Alarm,EO_CRON,ID,2,'Bad_data_version');
	END_IF
	SysFileClose(File:=hFile);
	RETURN;
END_IF

(* Read Jolly data *)
t2:=SysFileSetPos(File:=hFile, Pos:=512);
t1:=SysFileRead(File:=hFile, Buffer:=ADR(Jolly), Size:=SIZEOF(Jolly));
(* Read active profile index *)
CalendarIdx:=Sys.Time_CT_Day;
t2:=SysFileSetPos(File:=hFile, Pos:=(1024+4*CalendarIdx));
t1:=SysFileRead(File:=hFile, Buffer:=ADR(ProfileNr), Size:=SIZEOF(ProfileNr));
(* Read active profile *)
t2:=SysFileSetPos(File:=hFile, Pos:=(3072+512*ProfileNr));
t1:=SysFileRead(File:=hFile, Buffer:=ADR(Profile), Size:=SIZEOF(Profile));

(* Close file and validate data *)
SysFileClose(File:=hFile);
END_ACTION
ACTION DB_SetName:
(* Create current filename 'yyyyCRnn.DAT' *)
sFile:=CONCAT(FilesPath,WORD_TO_STRING(Sys.Time_Year));
sFile:=CONCAT(STR1:=sFile, STR2:='CR');
IF ID<10 THEN
sFile:=CONCAT(STR1:=sFile, STR2:='0');
END_IF
sFile:=CONCAT(STR1:=sFile, STR2:=BYTE_TO_STRING(ID));
sFile:=CONCAT(STR1:=sFile, STR2:='.DAT');
END_ACTION
ACTION Init:
DB_Load();
InitOK:=TRUE;
END_ACTION

(* POU Plant_Objects/obj_GATEWAY_01, ST *)
FUNCTION_BLOCK obj_GATEWAY_01
(* === ZIGBEE AMBIENT SENSORS MT-200 ===
   v1.0[07/05/05] - Create
*)
VAR CONSTANT
	LQI_Threshold		:	WORD := 100;		(* Zigbee link quality minimum value *)
	LowBattVoltage		:	WORD := 270;		(* Battery is considered low when reaches 1.35V each *)
END_VAR
VAR_INPUT
	(* Settings *)
	ID				: BYTE;
	Address			: BYTE;

(*	Refresh_Period	: TIME:=t#5m;
	(* Controls *)
	Refresh_Auto	: BOOL:=TRUE; (* Enable automatic refresh *)*)

	(* Modbus *)
	Refresh_Now	:	BOOL;	(* Start immediately modbus state machine *)
	retryErrMax	:	BYTE := 2;

	(* Limits *)
	Tmin			: INT := 50;
	Tmax			: INT := 400;
END_VAR
VAR_IN_OUT
	(* Interface *)
	ModBus		:obj_MODBUS;

END_VAR
VAR_OUTPUT
	(* Status *)
	Status_Log		: BYTE;
	Status_Vis 		: DWORD;
END_VAR
VAR


	state		:	INT;
	retry		:	BYTE;
	retryErr	:	BYTE;
	ReadTmr		:	TON := (PT:=T#5s);
	fModbusAlr:BOOL;


	AlarmCtr		: BYTE;
	WarningCtr		: BYTE;

	id_locale: BYTE;

	MB_RegistriLetti: ARRAY [0..40] OF WORD;

	Quality			: FLT_EVENT;
	Battery			: FLT_EVENT;
	Temperature		: FLT_EVENT := (INITEV:=FALSE);
	Alarm			: FLT_EVENT;

	ERR				: BOOL;
	fLQI			: BOOL;
	fBatt			: BOOL;
	fTemp			: BOOL;

	StatusOK		: BYTE;			(* 0: Status OK, >=1: Alarm and/or warning		Incremented by 1 when Alarm or Wrn occurs,
																					decremented by 1 when restored	*)
	TimeOutModBus: TON;
	ErroreComuModBus: BOOL;

	VerificaFuctionCode: INT;
	VerificaNodoLetto: INT;


END_VAR
(* stato creato per potere interrogare il nodo corretto *)
id_locale:=ID + 12;

Stm();
END_FUNCTION_BLOCK
ACTION Stm:
CASE state OF
	0:	(* Refresh time manager *)
		ReadTmr(IN:=NOT ReadTmr.Q);
		(*A tempo interrogo il nodo sempre che non ci sia qualcuno che lo sta interrogando in quel momento *)

		IF (ReadTmr.Q AND NodoDaInterrogareMB2=id_locale )OR Refresh_Now AND NOT InibiscoModbusMB2 THEN
			state := 10;
			ReadTmr.PT := T#5s;  (* moreno *)
			Refresh_Now := FALSE;
			InibiscoModbusMB2 := TRUE;
		END_IF

	(**** Leggo le Analogiche a Disposzione  ****)

	10:	(* richiedo lettura Holding Register   *)

		Modbus.MB_Query.SlaveAddress := Address;
		Modbus.MB_Query.FunctionCode := 4;
		ModBus.MB_Query.Read_StartAddress := 0 ;			(* richiedo lettura altri Parametri *)
		ModBus.MB_Query.Read_Quantity := 20;
		ModBus.MB_Start := TRUE;
		state := 20;

	20:	(* Risposta all'interrogazione *)
		IF NOT ModBus.MB_Start   THEN
			VerificaFuctionCode:=ModBus.MB_Resp.FunctionCode;
			VerificaNodoLetto:=ModBus.MB_Resp.SlaveAddress;

			IF ModBus.MB_MASTER.MB_Error<>0 THEN
				state := 300;
			ELSE

				MB_RegistriLetti[0] := ModBus.MB_Resp.Data[0];   	(* Vedi tabella *)
				MB_RegistriLetti[1] := ModBus.MB_Resp.Data[1];		(* Vedi tabella *)
				MB_RegistriLetti[2] := ModBus.MB_Resp.Data[2];		(* Vedi tabella *)
				MB_RegistriLetti[3] := ModBus.MB_Resp.Data[3];		(* Vedi tabella *)
				MB_RegistriLetti[4] := ModBus.MB_Resp.Data[4];		(* Vedi tabella *)
				MB_RegistriLetti[5] := ModBus.MB_Resp.Data[5];		(* Vedi tabella *)
				MB_RegistriLetti[6] := ModBus.MB_Resp.Data[6];		(* Vedi tabella *)
				MB_RegistriLetti[7] := ModBus.MB_Resp.Data[7];		(* Vedi tabella *)
				MB_RegistriLetti[8] := ModBus.MB_Resp.Data[8];		(* Vedi tabella *)
				MB_RegistriLetti[9] := ModBus.MB_Resp.Data[9];		(* Vedi tabella *)
				MB_RegistriLetti[10] := ModBus.MB_Resp.Data[10];		(* Vedi tabella *)
				MB_RegistriLetti[11] := ModBus.MB_Resp.Data[11];		(* Vedi tabella *)
				MB_RegistriLetti[12] := ModBus.MB_Resp.Data[12];		(* Vedi tabella *)
				MB_RegistriLetti[13] := ModBus.MB_Resp.Data[13];		(* Vedi tabella *)
				MB_RegistriLetti[14] := ModBus.MB_Resp.Data[14];		(* Vedi tabella *)
				MB_RegistriLetti[15] := ModBus.MB_Resp.Data[15];		(* Vedi tabella *)
				MB_RegistriLetti[16] := ModBus.MB_Resp.Data[16];		(* Vedi tabella *)
				MB_RegistriLetti[17] := ModBus.MB_Resp.Data[17];		(* Vedi tabella *)
				MB_RegistriLetti[18] := ModBus.MB_Resp.Data[18];		(* Vedi tabella *)
				MB_RegistriLetti[19] := ModBus.MB_Resp.Data[19];		(* Vedi tabella *)

				Modbus.MB_Query.SlaveAddress := Address;
				Modbus.MB_Query.FunctionCode := 4;
				ModBus.MB_Query.Read_StartAddress := 20 ;			(* richiedo lettura altri Parametri *)
				ModBus.MB_Query.Read_Quantity := 19;
				ModBus.MB_Start := TRUE;
				state := 30;

			END_IF
		END_IF

	30:	(* Risposta all'interrogazione *)
		IF NOT ModBus.MB_Start   THEN
			VerificaFuctionCode:=ModBus.MB_Resp.FunctionCode;
			VerificaNodoLetto:=ModBus.MB_Resp.SlaveAddress;

			IF ModBus.MB_MASTER.MB_Error<>0 THEN
				state := 300;
			ELSE

				MB_RegistriLetti[20] := ModBus.MB_Resp.Data[0];   	(* Vedi tabella *)
				MB_RegistriLetti[21] := ModBus.MB_Resp.Data[1];		(* Vedi tabella *)
				MB_RegistriLetti[22] := ModBus.MB_Resp.Data[2];		(* Vedi tabella *)
				MB_RegistriLetti[23] := ModBus.MB_Resp.Data[3];		(* Vedi tabella *)
				MB_RegistriLetti[24] := ModBus.MB_Resp.Data[4];		(* Vedi tabella *)
				MB_RegistriLetti[25] := ModBus.MB_Resp.Data[5];		(* Vedi tabella *)
				MB_RegistriLetti[26] := ModBus.MB_Resp.Data[6];		(* Vedi tabella *)
				MB_RegistriLetti[27] := ModBus.MB_Resp.Data[7];		(* Vedi tabella *)
				MB_RegistriLetti[28] := ModBus.MB_Resp.Data[8];		(* Vedi tabella *)
				MB_RegistriLetti[29] := ModBus.MB_Resp.Data[9];		(* Vedi tabella *)
				MB_RegistriLetti[30] := ModBus.MB_Resp.Data[10];		(* Vedi tabella *)
				MB_RegistriLetti[31] := ModBus.MB_Resp.Data[11];		(* Vedi tabella *)
				MB_RegistriLetti[32] := ModBus.MB_Resp.Data[12];		(* Vedi tabella *)
				MB_RegistriLetti[33] := ModBus.MB_Resp.Data[13];		(* Vedi tabella *)
				MB_RegistriLetti[34] := ModBus.MB_Resp.Data[14];		(* Vedi tabella *)
				MB_RegistriLetti[35] := ModBus.MB_Resp.Data[15];		(* Vedi tabella *)
				MB_RegistriLetti[36] := ModBus.MB_Resp.Data[16];		(* Vedi tabella *)
				MB_RegistriLetti[37] := ModBus.MB_Resp.Data[17];		(* Vedi tabella *)
				MB_RegistriLetti[38] := ModBus.MB_Resp.Data[18];		(* Vedi tabella *)
				MB_RegistriLetti[39] := ModBus.MB_Resp.Data[19];		(* Vedi tabella *)

				state := 295;

			END_IF
		END_IF






		295:
		IF NOT ModBus.MB_Start THEN
			IF ModBus.MB_MASTER.MB_Error<>0 THEN (*OR ModBus.MB_MASTER.MB_Error<>0 THEN*)
				state := 300;
			ELSE
				IF fModbusAlr THEN fModbusAlr := FALSE; END_IF
				NodoDaInterrogareMB2:=id_locale+1;
				InibiscoModbusMB2:=FALSE;
				retryErr := 0;
				retry := 0;
				state := 0;
					IF fModbusAlr=FALSE AND ErroreComuModBus=TRUE THEN
						LogEv(EL_Log,EO_CHI,ID,62,'ComunicazioneModBus_OK');
						ErroreComuModBus := FALSE;
				(*	WarningCtr := SEL(WarningCtr=0, WarningCtr-1, 0); *)
					END_IF


			END_IF
		END_IF



	(**** CHECK MODBUS ERROR ****)
	300: 	(* Release MODBUS *)
			InibiscoModbusMB3:=FALSE;
			(* Retries *)
			retry:=retry+1;
			IF retry>3 THEN
				retry:=0;

				(* Verify if slave is dead *)
				IF retryErr < retryErrMaX THEN
					retryErr := retryErr + 1;
				ELSE
					fModbusAlr := TRUE;
					(* Verify ModBus error	*)

					IF fModbusAlr AND ErroreComuModBus=FALSE THEN
						LogEv(EL_Alarm,EO_CHI,ID,61,CONCAT('ErroreModbus_',INT_TO_STRING(ModBus.MB_MASTER.MB_Error)));
						ErroreComuModBus := TRUE;
					END_IF
				END_IF

			END_IF
			Refresh_Now := FALSE;
			InibiscoModbusMB2:=FALSE;
			NodoDaInterrogareMB2:=id_locale+1;
			state:=0;
END_CASE




(* Controllo Time Out Ciclo ModBus *)

TimeOutModBus(In:=state<>0,PT:=t#30s);
IF TimeOutModBus.Q THEN
	State:=0;
	Refresh_Now:=TRUE;  (* Rilancio la lettura del nodo *)
	IF MODBUS.MB_Lock=TRUE THEN MODBUS.MB_Lock:=FALSE;END_IF
	IF InibiscoModbusMB2=TRUE THEN InibiscoModbusMB2:=FALSE;END_IF
END_IF
END_ACTION

(* POU Plant_Objects/obj_MODBUS_ANZFRER_01, ST *)
FUNCTION_BLOCK obj_MODBUS_ANZFRER_01
VAR CONSTANT

	TimeOutModBus: TON;


END_VAR
VAR_INPUT
	ID			:	BYTE;
	Address		:	BYTE;
	(* Modbus *)
	Refresh_Now	:	BOOL;			(* Richiesta di lettura stato macchina Immediata  *)
	retryErrMax	:	BYTE := 2;

(*	IndirizzoDaScrivere: WORD;
	DatoDaScrivere: INT;
	ScriviDato: BOOL; *)

END_VAR
VAR_IN_OUT
	ModBus		:obj_MODBUS;

END_VAR
VAR_OUTPUT
	Status_Log	:	WORD;
	Status_Vis	:	DWORD;
END_VAR
VAR

	state		:	INT;
	retry		:	BYTE;
	retryErr	:	BYTE;
	ReadTmr		:	TON := (PT:=T#5s);
	fModbusAlr:BOOL;

(*	retry_write	:	BYTE;
	fWriteStatus:	BOOL;
	fWriteMode	:	BOOL;
	fWriteReset	:	BOOL; *)

	x: INT;

	VerificaFuctionCode: INT;
	VerificaNodoLetto: INT;
	ErroreComuModBus: BOOL;
	IndiceErrore: BYTE;

	MB_BitStato: ARRAY [0..450] OF BOOL;
	MB_RegistriLetti: ARRAY [0..450] OF INT;




	AddressRead: BYTE;
	index: BYTE;
	indexErr: BYTE;


	MB_V_L1_N: DWORD;
	MB_V_L2_N: DWORD;
	MB_V_L3_N: DWORD;
	MB_V_L1_L2: DWORD;
	MB_V_L1_L3: DWORD;
	MB_V_L2_L3: DWORD;
	MB_V_IL1: DWORD;
	MB_V_IL2: DWORD;
	MB_V_IL3: DWORD;
	MB_V_F: DWORD;
	MB_V_P: DWORD;
	MB_V_Q: DWORD;
	MB_V_P_F: DWORD;
	MB_IL1_MAX: DWORD;
	MB_IL2_MAX: DWORD;
	MB_IL3_MAX: DWORD;
	MB_PF_IL1: DWORD;
	MB_PF_IL2: DWORD;
	MB_PF_IL3: DWORD;
	MB_COSPI_IL1: DWORD;
	MB_COSPI_IL2: DWORD;
	MB_COSPI_IL3: DWORD;
	MB_V_P_AVG: DWORD;
	MB_V_P_MAX: DWORD;
	MB_V_Q_MAX: DWORD;
	MB_V_Q_AVG: DWORD;
	MB_V_KWh: DWORD;
	MB_V_kVAr: DWORD;
	MB_Rappenergia: DWORD;


	moreno: ARRAY [0..20] OF WORD;

END_VAR
(* Call ModBus state machine *)
Stm();


(* Seganalzione stato Frigorifero  *)
IF ErroreComuModBus OR MB_BitStato[6] OR MB_BitStato[7] THEN
		Status_Log:=2; Status_Vis:=16#2020F0;
(*	ELSIF Warning OR Warning2 THEN
		Status_Log:=1; Status_Vis:=16#20F0F0; *)
    ELSE
		Status_Log:=0;
		Status_Vis:=16#006000;
END_IF
END_FUNCTION_BLOCK
ACTION AddLogData:
Logger.s1:=INSERT('&ANZ=',BYTE_TO_STRING(ID),4);
IF ID<10 THEN Logger.s1:=INSERT(Logger.s1,'0',4); END_IF


	Logger.s1:=CONCAT(Logger.s1,(REAL_TO_STRING(DWORD_TO_REAL(MB_V_L1_N)/1000)));
	Logger.s1:=CONCAT(Logger.s1,';');
	Logger.s1:=CONCAT(Logger.s1,(REAL_TO_STRING(DWORD_TO_REAL(MB_V_L2_N)/1000)));
	Logger.s1:=CONCAT(Logger.s1,';');
	Logger.s1:=CONCAT(Logger.s1,(REAL_TO_STRING(DWORD_TO_REAL(MB_V_L3_N)/1000)));
	Logger.s1:=CONCAT(Logger.s1,';');
	Logger.s1:=CONCAT(Logger.s1,(REAL_TO_STRING(DWORD_TO_REAL(MB_V_L1_L2)/1000)));
	Logger.s1:=CONCAT(Logger.s1,';');
	Logger.s1:=CONCAT(Logger.s1,(REAL_TO_STRING(DWORD_TO_REAL(MB_V_L1_L3)/1000)));
	Logger.s1:=CONCAT(Logger.s1,';');
	Logger.s1:=CONCAT(Logger.s1,(REAL_TO_STRING(DWORD_TO_REAL(MB_V_L2_L3)/1000)));
	Logger.s1:=CONCAT(Logger.s1,';');

	Logger.s1:=CONCAT(Logger.s1,(REAL_TO_STRING(DWORD_TO_REAL(MB_V_F))));
	Logger.s1:=CONCAT(Logger.s1,';');

	Logger.s1:=CONCAT(Logger.s1,(REAL_TO_STRING(DWORD_TO_REAL(MB_V_IL1))));
	Logger.s1:=CONCAT(Logger.s1,';');
	Logger.s1:=CONCAT(Logger.s1,(REAL_TO_STRING(DWORD_TO_REAL(MB_V_IL2))));
	Logger.s1:=CONCAT(Logger.s1,';');
	Logger.s1:=CONCAT(Logger.s1,(REAL_TO_STRING(DWORD_TO_REAL(MB_V_IL3))));
	Logger.s1:=CONCAT(Logger.s1,';');

	Logger.s1:=CONCAT(Logger.s1,(REAL_TO_STRING(DWORD_TO_REAL(MB_IL1_MAX))));
	Logger.s1:=CONCAT(Logger.s1,';');
	Logger.s1:=CONCAT(Logger.s1,(REAL_TO_STRING(DWORD_TO_REAL(MB_IL1_MAX))));
	Logger.s1:=CONCAT(Logger.s1,';');
	Logger.s1:=CONCAT(Logger.s1,(REAL_TO_STRING(DWORD_TO_REAL(MB_IL1_MAX))));
	Logger.s1:=CONCAT(Logger.s1,';');


	Logger.s1:=CONCAT(Logger.s1,(REAL_TO_STRING(DWORD_TO_REAL(MB_PF_IL1))));
	Logger.s1:=CONCAT(Logger.s1,';');
	Logger.s1:=CONCAT(Logger.s1,(REAL_TO_STRING(DWORD_TO_REAL(MB_PF_IL2))));
	Logger.s1:=CONCAT(Logger.s1,';');
	Logger.s1:=CONCAT(Logger.s1,(REAL_TO_STRING(DWORD_TO_REAL(MB_PF_IL3))));
	Logger.s1:=CONCAT(Logger.s1,';');

	Logger.s1:=CONCAT(Logger.s1,(REAL_TO_STRING(DWORD_TO_REAL(MB_V_P))));
	Logger.s1:=CONCAT(Logger.s1,';');
	Logger.s1:=CONCAT(Logger.s1,(REAL_TO_STRING(DWORD_TO_REAL(MB_V_P_AVG))));
	Logger.s1:=CONCAT(Logger.s1,';');
	Logger.s1:=CONCAT(Logger.s1,(REAL_TO_STRING(DWORD_TO_REAL(MB_V_P_MAX))));
	Logger.s1:=CONCAT(Logger.s1,';');

	Logger.s1:=CONCAT(Logger.s1,(REAL_TO_STRING(DWORD_TO_REAL(MB_V_Q))));
	Logger.s1:=CONCAT(Logger.s1,';');
	Logger.s1:=CONCAT(Logger.s1,(REAL_TO_STRING(DWORD_TO_REAL(MB_V_Q_MAX))));
	Logger.s1:=CONCAT(Logger.s1,';');


	CASE MB_Rappenergia OF
		1:	Logger.s1:=CONCAT(Logger.s1,(REAL_TO_STRING(DWORD_TO_REAL(MB_V_KWh)/100)));
			Logger.s1:=CONCAT(Logger.s1,';');
			Logger.s1:=CONCAT(Logger.s1,(REAL_TO_STRING(DWORD_TO_REAL(MB_V_kVAr)/100)));
			Logger.s1:=CONCAT(Logger.s1,';');

		10:	Logger.s1:=CONCAT(Logger.s1,(REAL_TO_STRING(DWORD_TO_REAL(MB_V_KWh)/10)));
			Logger.s1:=CONCAT(Logger.s1,';');
			Logger.s1:=CONCAT(Logger.s1,(REAL_TO_STRING(DWORD_TO_REAL(MB_V_kVAr)/10)));
			Logger.s1:=CONCAT(Logger.s1,';');

		100:Logger.s1:=CONCAT(Logger.s1,(REAL_TO_STRING(DWORD_TO_REAL(MB_V_KWh))));
			Logger.s1:=CONCAT(Logger.s1,';');
			Logger.s1:=CONCAT(Logger.s1,(REAL_TO_STRING(DWORD_TO_REAL(MB_V_kVAr))));
			Logger.s1:=CONCAT(Logger.s1,';');

	END_CASE

	Logger.s1:=CONCAT(Logger.s1,WORD_TO_STRING(Status_Log));
	Logger.s1:=CONCAT(Logger.s1,';');

	Logger.s1:=CONCAT(Logger.s1,(REAL_TO_STRING(DWORD_TO_REAL(MB_COSPI_IL1))));
	Logger.s1:=CONCAT(Logger.s1,';');
	Logger.s1:=CONCAT(Logger.s1,(REAL_TO_STRING(DWORD_TO_REAL(MB_COSPI_IL2))));
	Logger.s1:=CONCAT(Logger.s1,';');
	Logger.s1:=CONCAT(Logger.s1,(REAL_TO_STRING(DWORD_TO_REAL(MB_COSPI_IL3))));
	Logger.s1:=CONCAT(Logger.s1,';');
	Logger.s1:=CONCAT(Logger.s1,'0');    (* 0=3-phase, 1 = mono phase *)


ADDSTRING(ADR(Logger.TData), ADR(Logger.s1), Logger.TLen);
END_ACTION
ACTION Stm:
CASE state OF
	0:	(* Refresh time manager *)
		ReadTmr(IN:=NOT ReadTmr.Q);
		(*A tempo interrogo il nodo sempre che non ci sia qualcuno che lo sta interrogando in quel momento *)

		IF (ReadTmr.Q AND NodoDaInterrogareANZ=Address )OR Refresh_Now AND NOT InibiscoModbusANZ THEN
			state := 10;
			ReadTmr.PT := T#5s;
			Refresh_Now := FALSE;
			InibiscoModbusANZ := TRUE;
		END_IF

	(**** Leggo le Analogiche a Disposzione  ****)

	10:	(* richiedo lettura Holding Registere Chiller  *)

		Modbus.MB_Query.SlaveAddress := Address;
		Modbus.MB_Query.FunctionCode := 3;
		ModBus.MB_Query.Read_StartAddress := 256 ;			(* richiedo lettura altri Parametri *)
		ModBus.MB_Query.Read_Quantity := 20;
		ModBus.MB_Start := TRUE;
		state := 20;

	20:	(* Risposta all'interrogazione *)
		IF NOT ModBus.MB_Start   THEN
			VerificaFuctionCode:=ModBus.MB_Resp.FunctionCode;
			VerificaNodoLetto:=ModBus.MB_Resp.SlaveAddress;

			IF ModBus.MB_MASTER.MB_Error<>0 THEN
				state := 300;
			ELSE
				MB_V_L1_N:= ModBus.MB_Resp.Data[0]*65536 +  ModBus.MB_Resp.Data[1];   	(* Vedi tabella *)
				MB_V_L2_N:= ModBus.MB_Resp.Data[2]*65536 +  ModBus.MB_Resp.Data[3];   	(* Vedi tabella *)
				MB_V_L3_N:= ModBus.MB_Resp.Data[4]*65536 +  ModBus.MB_Resp.Data[5];   	(* Vedi tabella *)
				MB_V_L1_L2:= ModBus.MB_Resp.Data[6]*65536 +  ModBus.MB_Resp.Data[7];   	(* Vedi tabella *)
				MB_V_L1_L3:= ModBus.MB_Resp.Data[8]*65536 +  ModBus.MB_Resp.Data[9];   	(* Vedi tabella *)
				MB_V_L2_L3:= ModBus.MB_Resp.Data[10]*65536 +  ModBus.MB_Resp.Data[11];   	(* Vedi tabella *)
				ModBus.MB_Query.Read_StartAddress := 268; 	(* richiedo lettura altri Parametri *)
				ModBus.MB_Query.Read_Quantity := 10;
				ModBus.MB_Start := TRUE;

				state := 30;
			END_IF
		END_IF

	30: (* Rispota Altri paramenti *)
		IF NOT ModBus.MB_Start  THEN

			IF ModBus.MB_MASTER.MB_Error<>0 THEN
				state := 300;
			ELSE
				MB_V_IL1:= ModBus.MB_Resp.Data[0]*65536 +  ModBus.MB_Resp.Data[1];   	(* Vedi tabella *)
				MB_V_IL2:= ModBus.MB_Resp.Data[2]*65536 +  ModBus.MB_Resp.Data[3];   	(* Vedi tabella *)
				MB_V_IL3:= ModBus.MB_Resp.Data[4]*65536 +  ModBus.MB_Resp.Data[5];   	(* Vedi tabella *)
				MB_V_F:= ModBus.MB_Resp.Data[6]*65536 +  ModBus.MB_Resp.Data[7];   	(* Vedi tabella *)
				MB_V_P:= ModBus.MB_Resp.Data[8]*65536 +  ModBus.MB_Resp.Data[9];   	(* Vedi tabella *)

				ModBus.MB_Query.Read_StartAddress := 278; (* richiedo lettura altri Parametri *)
				ModBus.MB_Query.Read_Quantity := 20;
				ModBus.MB_Start := TRUE;

				state := 40;
			END_IF
		END_IF



	40: (* Rispota Altri paramenti *)
		IF NOT ModBus.MB_Start  THEN

			IF ModBus.MB_MASTER.MB_Error<>0 THEN
				state := 300;
			ELSE
				MB_V_Q:= ModBus.MB_Resp.Data[0]*65536 +  ModBus.MB_Resp.Data[1];   	(* Vedi tabella *)
				MB_V_P_F:= ModBus.MB_Resp.Data[2]*65536 +  ModBus.MB_Resp.Data[3];   	(* Vedi tabella *)
				MB_V_KWh:= ModBus.MB_Resp.Data[4]*65536 +  ModBus.MB_Resp.Data[5];   	(* Vedi tabella *)
				MB_V_kVAr:= ModBus.MB_Resp.Data[6]*65536 +  ModBus.MB_Resp.Data[7];   	(* Vedi tabella *)
				MB_Rappenergia:= ModBus.MB_Resp.Data[8]*65536 +  ModBus.MB_Resp.Data[9];   	(* Vedi tabella *)

				ModBus.MB_Query.Read_StartAddress := 354; (* richiedo lettura altri Parametri *)
				ModBus.MB_Query.Read_Quantity := 20;
				ModBus.MB_Start := TRUE;

				state := 50;
			END_IF
		END_IF

	50: (* Rispota Altri paramenti *)
		IF NOT ModBus.MB_Start  THEN

			IF ModBus.MB_MASTER.MB_Error<>0 THEN
				state := 300;
			ELSE

				MB_V_P_AVG:= ModBus.MB_Resp.Data[0]*65536 +  ModBus.MB_Resp.Data[1];   	(* Vedi tabella *)
				MB_V_P_MAX:= ModBus.MB_Resp.Data[2]*65536 +  ModBus.MB_Resp.Data[3];   	(* Vedi tabella *)
				MB_IL1_MAX:= ModBus.MB_Resp.Data[4]*65536 +  ModBus.MB_Resp.Data[5];   	(* Vedi tabella *)
				MB_IL2_MAX:= ModBus.MB_Resp.Data[6]*65536 +  ModBus.MB_Resp.Data[7];   	(* Vedi tabella *)
				MB_IL3_MAX:= ModBus.MB_Resp.Data[8]*65536 +  ModBus.MB_Resp.Data[9];   	(* Vedi tabella *)

				ModBus.MB_Query.Read_StartAddress := 342; (* richiedo lettura altri Parametri *)
				ModBus.MB_Query.Read_Quantity := 20;
				ModBus.MB_Start := TRUE;

				state := 55;
			END_IF
		END_IF

	55: (* Rispota Altri paramenti *)
		IF NOT ModBus.MB_Start  THEN

			IF ModBus.MB_MASTER.MB_Error<>0 THEN
				state := 300;
			ELSE
				MB_PF_IL1:= ModBus.MB_Resp.Data[0]*65536 +  ModBus.MB_Resp.Data[1];   	(* Vedi tabella *)
				MB_PF_IL2:= ModBus.MB_Resp.Data[2]*65536 +  ModBus.MB_Resp.Data[3];   	(* Vedi tabella *)
				MB_PF_IL3:= ModBus.MB_Resp.Data[4]*65536 +  ModBus.MB_Resp.Data[5];   	(* Vedi tabella *)
				MB_COSPI_IL1:= ModBus.MB_Resp.Data[6]*65536 +  ModBus.MB_Resp.Data[7];   	(* Vedi tabella *)
				MB_COSPI_IL2:= ModBus.MB_Resp.Data[8]*65536 +  ModBus.MB_Resp.Data[9];   	(* Vedi tabella *)
				MB_COSPI_IL3:= ModBus.MB_Resp.Data[10]*65536 +  ModBus.MB_Resp.Data[11];   	(* Vedi tabella *)

				ModBus.MB_Query.Read_StartAddress := 422; (* richiedo lettura altri Parametri *)
				ModBus.MB_Query.Read_Quantity := 20;
				ModBus.MB_Start := TRUE;

				state := 60;
			END_IF
		END_IF

	60: (* Rispota Altri paramenti *)
		IF NOT ModBus.MB_Start  THEN

			IF ModBus.MB_MASTER.MB_Error<>0 THEN
				state := 300;
			ELSE
				MB_V_Q_MAX:= ModBus.MB_Resp.Data[0]*65536 +  ModBus.MB_Resp.Data[1];   	(* Vedi tabella *)
				MB_V_Q_AVG:= ModBus.MB_Resp.Data[2]*65536 +  ModBus.MB_Resp.Data[3];   	(* Vedi tabella *)

				(* ModBus.MB_Query.Read_StartAddress := 422; (* richiedo lettura altri Parametri *)
				ModBus.MB_Query.Read_Quantity := 20;
				ModBus.MB_Start := TRUE; *)

				state := 295;
			END_IF
		END_IF





		295:
		IF NOT ModBus.MB_Start THEN
			IF ModBus.MB_MASTER.MB_Error<>0 THEN (*OR ModBus.MB_MASTER.MB_Error<>0 THEN*)
				state := 300;
			ELSE
				IF fModbusAlr THEN fModbusAlr := FALSE; END_IF
				NodoDaInterrogareANZ:=Address+1;
				InibiscoModbusANZ:=FALSE;
				retryErr := 0;
				retry := 0;
				state := 0;
					IF fModbusAlr=FALSE AND ErroreComuModBus=TRUE THEN
						LogEv(EL_Log,EO_CHI,ID,62,'ComunicazioneModBus_OK');
						ErroreComuModBus := FALSE;
				(*	WarningCtr := SEL(WarningCtr=0, WarningCtr-1, 0); *)
					END_IF


			END_IF
		END_IF



	(**** CHECK MODBUS ERROR ****)
	300: 	(* Release MODBUS *)
			InibiscoModbusANZ:=FALSE;
			(* Retries *)
			retry:=retry+1;
			IF retry>3 THEN
				retry:=0;

				(* Verify if slave is dead *)
				IF retryErr < retryErrMaX THEN
					retryErr := retryErr + 1;
				ELSE
					fModbusAlr := TRUE;
					(* Verify ModBus error	*)

					IF fModbusAlr AND ErroreComuModBus=FALSE THEN
						LogEv(EL_Alarm,EO_CHI,ID,61,CONCAT('ErroreModbus_',INT_TO_STRING(ModBus.MB_MASTER.MB_Error)));
						ErroreComuModBus := TRUE;
					END_IF
				END_IF

				END_IF
			Refresh_Now := FALSE;
			InibiscoModbusANZ:=FALSE;
			NodoDaInterrogareANZ:=Address+1;
			state:=0;
END_CASE




(* Controllo Time Out Ciclo ModBus *)

TimeOutModBus(In:=state<>0,PT:=t#30s);
IF TimeOutModBus.Q THEN
	State:=0;
	Refresh_Now:=TRUE;  (* Rilancio la lettura del nodo *)
	IF MODBUS.MB_Lock=TRUE THEN MODBUS.MB_Lock:=FALSE;END_IF
	IF InibiscoModbusANZ=TRUE THEN InibiscoModbusANZ:=FALSE;END_IF
END_IF
END_ACTION

(* POU Plant_Objects/obj_MODBUS_FRG_AER485P1, ST *)
FUNCTION_BLOCK obj_MODBUS_FRG_AER485P1
VAR CONSTANT

	TimeOutModBus: TON;


END_VAR
VAR_INPUT
	ID			:	BYTE;
	Address		:	BYTE;


	SetPointManuale: INT; 			(* SetPoint forazato in manuale escludendo la curva di carico *)
	AbilitaSetPointManuale : BOOL ; (* Abilita il funzionamento col set point Manaule Escludendo la curva cliamtica *)


	(* Modbus *)
	Refresh_Now	:	BOOL;			(* Richiesta di lettura stato macchina Immediata  *)
	retryErrMax	:	BYTE := 2;

	Temperatura: INT;


	STOP_REQ: BOOL;
	RUN_REQ: BOOL;
	(* Timings *)
	OnDelay		:	TIME;
	OffDelay	:	TIME;

	OnOff		: 	BOOL;

	IndirizzoDaScrivere: WORD;
	DatoDaScrivere: INT;
	ScriviDato: BOOL;
	ScriviCoil: BOOL;


	ImpMB_2SetPoint: INT;
	ImpMB_ResetFrigo: BOOL;
	ImpMB_LocRem: BOOL;
	fWriteAttivazioneComandi:BOOL;




END_VAR
VAR_IN_OUT
	ModBus		:obj_MODBUS;
	CLIM		:typ_Clima;

END_VAR
VAR_OUTPUT
	Run			:	BOOL;

	Status_Log	:	WORD;
	Status_Vis	:	DWORD;
END_VAR
VAR
	(* da diego per gestione stato stringa > 255*)
	temp :STRING(255);
	tempRaw		: ARRAY [0..MAX_SEND_TCP_CLIENT] OF BYTE;
	tempRawLen :DINT;
	longString:STRING(800);

	(* Timer manage switch on/off delay *)
	Delay		: 	TONOF;

	AllarmeFrigo_MB		:ARRAY [0..100] OF	FLT_EVENT;
	Warning		:	FLT_TAP := (TAP:=100);

	state		:	INT;
	retry		:	BYTE;
	retryErr	:	BYTE;
	ReadTmr		:	TON := (PT:=T#5s);
	fModbusAlr:BOOL;

(*	retry_write	:	BYTE;
	fWriteStatus:	BOOL;
	fWriteMode	:	BOOL;
	fWriteReset	:	BOOL; *)

	SetPointCC: DINT;
	x: INT;
	ImpMB_SetPoint: INT;
	Ctrl_Run: BOOL;


	VerificaFuctionCode: INT;
	VerificaNodoLetto: INT;
	ErroreComuModBus: BOOL;
	IndiceErrore: BYTE;

	MB_BitStato: ARRAY [0..200] OF BOOL;
	MB_RegistriLetti: ARRAY [0..450] OF INT;


	AddressRead: BYTE;
	index: BYTE;
	indexErr: BYTE;





END_VAR
VAR_INPUT RETAIN
	ChillerAbilitato: BOOL;
END_VAR
(* Aggiornamento in tempo reale dei TON e TOFF funzionamento Pompa *)

Delay.PT_OF := OffDelay;
Delay.PT_ON := OnDelay + WORD_TO_TIME(1000*ID);

(* Check climatic setup *)
IF NOT CLIM.InitOK THEN Clima_Default(); END_IF;
(* Calculate Setpoint *)

	IF Temperatura>=CLIM.Points[0].X  THEN SetPointCC:=CLIM.Points[0].Y; END_IF;
	IF Temperatura>=CLIM.Points[1].X AND Temperatura<CLIM.Points[0].X THEN SetPointCC:=CLIM.Points[0].Y; END_IF;
	IF Temperatura>=CLIM.Points[2].X AND Temperatura<CLIM.Points[1].X THEN SetPointCC:=CLIM.Points[1].Y; END_IF;
	IF Temperatura>=CLIM.Points[3].X AND Temperatura<CLIM.Points[2].X THEN SetPointCC:=CLIM.Points[2].Y; END_IF;
	IF Temperatura>=CLIM.Points[4].X AND Temperatura<CLIM.Points[3].X THEN SetPointCC:=CLIM.Points[3].Y; END_IF;
	IF Temperatura<CLIM.Points[4].X THEN SetPointCC:=CLIM.Points[4].Y; END_IF;


	IF Temperatura<CLIM.Points[4].X THEN SetPointCC:=CLIM.Points[4].Y; END_IF;


(* Scelta del set point della cladaia o vien preso dalla curva cliamtica o da un riferimento esterno *)
IF AbilitaSetPointManuale THEN
	ImpMB_SetPoint:=(SetPointManuale);
ELSE
	ImpMB_SetPoint:=DINT_TO_INT(SetPointCC);
END_IF


(* Controllo Bit di funzionamento ON e OFF  *)
Ctrl_Run := OnOff AND ChillerAbilitato;
Delay(IN:=Ctrl_Run);



IF STOP_REQ THEN Run := 1;
	ELSIF RUN_REQ THEN Run := 0;
ELSE
	Run :=Delay.OUT AND ChillerAbilitato;
END_IF



(* Call ModBus state machine *)
Stm();

(* Check alarm	*)
CheckAlarm();



(* Seganalzione stato Frigorifero  *)
IF ErroreComuModBus OR MB_BitStato[6] OR MB_BitStato[7] THEN
		Status_Log:=2; Status_Vis:=16#2020F0;
(*	ELSIF Warning OR Warning2 THEN
		Status_Log:=1; Status_Vis:=16#20F0F0; *)
    ELSE
		Status_Log:=0;
		Status_Vis:=16#006000;
END_IF
END_FUNCTION_BLOCK
ACTION AddLogData:
Logger.s1:=INSERT('&CHIAERMEC=',BYTE_TO_STRING(ID),10);
IF ID<10 THEN Logger.s1:=INSERT(Logger.s1,'0',10); END_IF

FOR tempRawLen:=0 TO MAX_SEND_TCP_CLIENT DO
                tempRaw[tempRawLen]:=0;
END_FOR

tempRawLen:=0;


temp:=Logger.s1;
ADDSTRING(ADR(tempRaw), ADR(temp), tempRawLen);

FOR x:= 1 TO 2 DO

	temp:=CONCAT(INT_TO_STRING(MB_RegistriLetti[x]),';');
	ADDSTRING(ADR(tempRaw), ADR(temp), tempRawLen);

END_FOR


FOR x:= 5 TO 15 DO
	temp:=CONCAT(INT_TO_STRING(MB_RegistriLetti[x]),';');
	ADDSTRING(ADR(tempRaw), ADR(temp), tempRawLen);
END_FOR

FOR x:= 21 TO 23 DO
	temp:=CONCAT(INT_TO_STRING(MB_RegistriLetti[x]),';');
	ADDSTRING(ADR(tempRaw), ADR(temp), tempRawLen);
END_FOR

FOR x:= 25 TO 25 DO
	temp:=CONCAT(INT_TO_STRING(MB_RegistriLetti[x]),';');
	ADDSTRING(ADR(tempRaw), ADR(temp), tempRawLen);
END_FOR


FOR x:= 180 TO 181 DO
	temp:=CONCAT(INT_TO_STRING(MB_RegistriLetti[x]),';');
	ADDSTRING(ADR(tempRaw), ADR(temp), tempRawLen);
END_FOR

FOR x:= 184 TO 186 DO
	temp:=CONCAT(INT_TO_STRING(MB_RegistriLetti[x]),';');
	ADDSTRING(ADR(tempRaw), ADR(temp), tempRawLen);
END_FOR

FOR x:= 189 TO 207 DO
	temp:=CONCAT(INT_TO_STRING(MB_RegistriLetti[x]),';');
	ADDSTRING(ADR(tempRaw), ADR(temp), tempRawLen);
END_FOR

FOR x:= 209 TO 215 DO
	temp:=CONCAT(INT_TO_STRING(MB_RegistriLetti[x]),';');
	ADDSTRING(ADR(tempRaw), ADR(temp), tempRawLen);
END_FOR

FOR x:= 218 TO 219 DO
	temp:=CONCAT(INT_TO_STRING(MB_RegistriLetti[x]),';');
	ADDSTRING(ADR(tempRaw), ADR(temp), tempRawLen);
END_FOR

FOR x:= 232 TO 232 DO
	temp:=CONCAT(INT_TO_STRING(MB_RegistriLetti[x]),';');
	ADDSTRING(ADR(tempRaw), ADR(temp), tempRawLen);
END_FOR

FOR x:= 235 TO 238 DO
	temp:=CONCAT(INT_TO_STRING(MB_RegistriLetti[x]),';');
	ADDSTRING(ADR(tempRaw), ADR(temp), tempRawLen);
END_FOR

FOR x:= 408 TO 413 DO
	temp:=CONCAT(INT_TO_STRING(MB_RegistriLetti[x]),';');
	ADDSTRING(ADR(tempRaw), ADR(temp), tempRawLen);
END_FOR

FOR x:= 1 TO 19 DO
	temp:=CONCAT(SEL(MB_BitStato[x],'0','1'),';');
	ADDSTRING(ADR(tempRaw), ADR(temp), tempRawLen);
END_FOR

	temp:=CONCAT(SEL(MB_BitStato[21],'0','1'),';');
	ADDSTRING(ADR(tempRaw), ADR(temp), tempRawLen);

FOR x:= 28 TO 31 DO
	temp:=CONCAT(SEL(MB_BitStato[x],'0','1'),';');
	ADDSTRING(ADR(tempRaw), ADR(temp), tempRawLen);
END_FOR

FOR x:= 34 TO 59 DO
	temp:=CONCAT(SEL(MB_BitStato[x],'0','1'),';');
	ADDSTRING(ADR(tempRaw), ADR(temp), tempRawLen);
END_FOR

FOR x:= 100 TO 104 DO
	temp:=CONCAT(SEL(MB_BitStato[x],'0','1'),';');
	ADDSTRING(ADR(tempRaw), ADR(temp), tempRawLen);
END_FOR

FOR x:= 107 TO 117 DO
	temp:=CONCAT(SEL(MB_BitStato[x],'0','1'),';');
	ADDSTRING(ADR(tempRaw), ADR(temp), tempRawLen);
END_FOR

FOR x:= 119 TO 131 DO
	temp:=CONCAT(SEL(MB_BitStato[x],'0','1'),';');
	ADDSTRING(ADR(tempRaw), ADR(temp), tempRawLen);
END_FOR

FOR x:= 134 TO 151 DO
	temp:=CONCAT(SEL(MB_BitStato[x],'0','1'),';');
	ADDSTRING(ADR(tempRaw), ADR(temp), tempRawLen);
END_FOR


temp:=CONCAT(SEL(MB_BitStato[153],'0','1'),';');
ADDSTRING(ADR(tempRaw), ADR(temp), tempRawLen);
temp:=CONCAT(SEL(MB_BitStato[154],'0','1'),';');
ADDSTRING(ADR(tempRaw), ADR(temp), tempRawLen);


FOR x:= 158 TO 164 DO
	temp:=CONCAT(SEL(MB_BitStato[x],'0','1'),';');
	ADDSTRING(ADR(tempRaw), ADR(temp), tempRawLen);
END_FOR

temp:=CONCAT(SEL(MB_BitStato[166],'0','1'),';');
ADDSTRING(ADR(tempRaw), ADR(temp), tempRawLen);


FOR x:= 168 TO 178 DO
	temp:=CONCAT(SEL(MB_BitStato[x],'0','1'),';');
	ADDSTRING(ADR(tempRaw), ADR(temp), tempRawLen);
END_FOR


FOR x:= 180 TO 198 DO
	temp:=CONCAT(SEL(MB_BitStato[x],'0','1'),';');
	ADDSTRING(ADR(tempRaw), ADR(temp), tempRawLen);
END_FOR

temp:=SEL(MB_BitStato[199],'0','1');

ADDSTRING(ADR(tempRaw), ADR(temp), tempRawLen);

ADDSTRING(ADR(Logger.TData), ADR(tempRaw), Logger.TLen);
END_ACTION
ACTION CheckAlarm:
(**** GEstione Log ad Evento *****)


FOR x:=0 TO 100 DO

	AllarmeFrigo_MB[x](IN:=MB_BitStato[x+100] );

	IF AllarmeFrigo_MB[x].EVH THEN
		LogEv(EL_Alarm,EO_CHIAERMEC,ID,1,CONCAT ('AllarmeAttivo_n.', INT_TO_STRING(x+100)));
(*		LogEv(EL_Alarm,EO_CHIAERMEC,ID,x+100,CONCAT ('Allarme Attivo n. ', INT_TO_STRING(x+100))); *)
	END_IF

	IF AllarmeFrigo_MB[x].EVL THEN
		LogEv(EL_Log,EO_CHIAERMEC,ID,2,CONCAT ('AllarmeRientrato_n.', INT_TO_STRING(x+100)));
(*		LogEv(EL_Log,EO_CHIAERMEC,ID,x+100,CONCAT ('Allarme Rientrato n. ', INT_TO_STRING(x+100))); *)
	END_IF

END_FOR
END_ACTION
ACTION Clima_Default:
IF CLIM.Points[0].X=0 THEN
	CLIM.Points[0].X:=-300; CLIM.Points[0].Y:=770;
	CLIM.Points[1].X:=-70 ; CLIM.Points[1].Y:=770;
	CLIM.Points[2].X:= 80; 	CLIM.Points[2].Y:=690;
	CLIM.Points[3].X:= 200; CLIM.Points[3].Y:=300;
	CLIM.Points[4].X:= 500; CLIM.Points[4].Y:=200;
END_IF
CLIM.InitOK:=TRUE;
LogEv(EL_Wrn,EO_chi,ID,0,'Climatic_default');
END_ACTION
ACTION Stm:
CASE state OF
	0:	(* Refresh time manager *)
		ReadTmr(IN:=NOT ReadTmr.Q);
		(*A tempo interrogo il nodo sempre che non ci sia qualcuno che lo sta interrogando in quel momento *)

		IF (ReadTmr.Q AND NodoDaInterrogareChiller=Address )OR Refresh_Now AND NOT InibiscoModbusChiller THEN
			state := 10;
			ReadTmr.PT := T#5s;  (* moreno *)
			Refresh_Now := FALSE;
			InibiscoModbusChiller := TRUE;
		END_IF

	(**** Leggo le Analogiche a Disposzione  ****)

	10:	(* richiedo lettura Holding Registere Chiller  *)

		Modbus.MB_Query.SlaveAddress := Address;
		Modbus.MB_Query.FunctionCode := 3;
		ModBus.MB_Query.Read_StartAddress := 0 ;			(* richiedo lettura altri Parametri *)
		ModBus.MB_Query.Read_Quantity := 3;
		ModBus.MB_Start := TRUE;
		state := 20;

	20:	(* Risposta all'interrogazione *)
		IF NOT ModBus.MB_Start   THEN
			VerificaFuctionCode:=ModBus.MB_Resp.FunctionCode;
			VerificaNodoLetto:=ModBus.MB_Resp.SlaveAddress;

			IF ModBus.MB_MASTER.MB_Error<>0 THEN
				state := 300;
			ELSE
				MB_RegistriLetti[0] := ModBus.MB_Resp.Data[0];   	(* Vedi tabella *)
				MB_RegistriLetti[1] := ModBus.MB_Resp.Data[1];		(* Vedi tabella *)
				MB_RegistriLetti[2] := ModBus.MB_Resp.Data[2];		(* Vedi tabella *)


				ModBus.MB_Query.Read_StartAddress := 5; 	(* richiedo lettura altri Parametri *)
				ModBus.MB_Query.Read_Quantity := 11;
				ModBus.MB_Start := TRUE;

				state := 30;
			END_IF
		END_IF

	30: (* Rispota Altri paramenti *)
		IF NOT ModBus.MB_Start  THEN

			IF ModBus.MB_MASTER.MB_Error<>0 THEN
				state := 300;
			ELSE
				MB_RegistriLetti[5] := ModBus.MB_Resp.Data[0];   	(* Vedi tabella *)
				MB_RegistriLetti[6] := ModBus.MB_Resp.Data[1];		(* Vedi tabella *)
				MB_RegistriLetti[7] := ModBus.MB_Resp.Data[2];		(* Vedi tabella *)
				MB_RegistriLetti[8] := ModBus.MB_Resp.Data[3];		(* Vedi tabella *)
				MB_RegistriLetti[9] := ModBus.MB_Resp.Data[4];		(* Vedi tabella *)
				MB_RegistriLetti[10] := ModBus.MB_Resp.Data[5];		(* Vedi tabella *)
				MB_RegistriLetti[11] := ModBus.MB_Resp.Data[6];		(* Vedi tabella *)
				MB_RegistriLetti[12] := ModBus.MB_Resp.Data[7];		(* Vedi tabella *)
				MB_RegistriLetti[13] := ModBus.MB_Resp.Data[8];		(* Vedi tabella *)
				MB_RegistriLetti[14] := ModBus.MB_Resp.Data[9];		(* Vedi tabella *)
				MB_RegistriLetti[15] := ModBus.MB_Resp.Data[10];		(* Vedi tabella *)

				ModBus.MB_Query.Read_StartAddress := 21; (* richiedo lettura altri Parametri *)
				ModBus.MB_Query.Read_Quantity := 5;
				ModBus.MB_Start := TRUE;

				state := 40;
			END_IF
		END_IF

	40: (* Rispota Altri paramenti *)
		IF NOT ModBus.MB_Start  THEN

			IF ModBus.MB_MASTER.MB_Error<>0 THEN
				state := 300;
			ELSE
				MB_RegistriLetti[21] := ModBus.MB_Resp.Data[0];   	(* Vedi tabella *)
				MB_RegistriLetti[22] := ModBus.MB_Resp.Data[1];		(* Vedi tabella *)
				MB_RegistriLetti[23] := ModBus.MB_Resp.Data[2];		(* Vedi tabella *)
				MB_RegistriLetti[24] := ModBus.MB_Resp.Data[3];		(* Vedi tabella *)
				MB_RegistriLetti[25] := ModBus.MB_Resp.Data[4];		(* Vedi tabella *)

				ModBus.MB_Query.Read_StartAddress := 180; (* richiedo lettura altri Parametri *)
				ModBus.MB_Query.Read_Quantity := 20;
				ModBus.MB_Start := TRUE;

				state := 45;
			END_IF
		END_IF

	45: (* Rispota Altri paramenti *)
		IF NOT ModBus.MB_Start  THEN

			IF ModBus.MB_MASTER.MB_Error<>0 THEN
				state := 300;
			ELSE
				MB_RegistriLetti[180] := ModBus.MB_Resp.Data[0];   	(* Vedi tabella *)
				MB_RegistriLetti[181] := ModBus.MB_Resp.Data[1];		(* Vedi tabella *)
				MB_RegistriLetti[182] := ModBus.MB_Resp.Data[2];		(* Vedi tabella *)
				MB_RegistriLetti[183] := ModBus.MB_Resp.Data[3];		(* Vedi tabella *)
				MB_RegistriLetti[184] := ModBus.MB_Resp.Data[4];		(* Vedi tabella *)
				MB_RegistriLetti[185] := ModBus.MB_Resp.Data[5];		(* Vedi tabella *)
				MB_RegistriLetti[186] := ModBus.MB_Resp.Data[6];		(* Vedi tabella *)
				MB_RegistriLetti[187] := ModBus.MB_Resp.Data[7];		(* Vedi tabella *)
				MB_RegistriLetti[188] := ModBus.MB_Resp.Data[8];		(* Vedi tabella *)
				MB_RegistriLetti[189] := ModBus.MB_Resp.Data[9];		(* Vedi tabella *)
				MB_RegistriLetti[190] := ModBus.MB_Resp.Data[10];		(* Vedi tabella *)
				MB_RegistriLetti[191] := ModBus.MB_Resp.Data[11];		(* Vedi tabella *)
				MB_RegistriLetti[192] := ModBus.MB_Resp.Data[12];		(* Vedi tabella *)
				MB_RegistriLetti[193] := ModBus.MB_Resp.Data[13];		(* Vedi tabella *)
				MB_RegistriLetti[194] := ModBus.MB_Resp.Data[14];		(* Vedi tabella *)
				MB_RegistriLetti[195] := ModBus.MB_Resp.Data[15];		(* Vedi tabella *)
				MB_RegistriLetti[196] := ModBus.MB_Resp.Data[16];		(* Vedi tabella *)
				MB_RegistriLetti[197] := ModBus.MB_Resp.Data[17];		(* Vedi tabella *)
				MB_RegistriLetti[198] := ModBus.MB_Resp.Data[18];		(* Vedi tabella *)
				MB_RegistriLetti[199] := ModBus.MB_Resp.Data[19];		(* Vedi tabella *)

				ModBus.MB_Query.Read_StartAddress := 200; (* richiedo lettura altri Parametri *)
				ModBus.MB_Query.Read_Quantity := 9;
				ModBus.MB_Start := TRUE;

				state := 50;
			END_IF
		END_IF
	50: (* Rispota Altri paramenti *)
		IF NOT ModBus.MB_Start  THEN

			IF ModBus.MB_MASTER.MB_Error<>0 THEN
				state := 300;
			ELSE
				MB_RegistriLetti[200] := ModBus.MB_Resp.Data[0];   	(* Vedi tabella *)
				MB_RegistriLetti[201] := ModBus.MB_Resp.Data[1];		(* Vedi tabella *)
				MB_RegistriLetti[202] := ModBus.MB_Resp.Data[2];		(* Vedi tabella *)
				MB_RegistriLetti[203] := ModBus.MB_Resp.Data[3];		(* Vedi tabella *)
				MB_RegistriLetti[204] := ModBus.MB_Resp.Data[4];		(* Vedi tabella *)
				MB_RegistriLetti[205] := ModBus.MB_Resp.Data[5];		(* Vedi tabella *)
				MB_RegistriLetti[206] := ModBus.MB_Resp.Data[6];		(* Vedi tabella *)
				MB_RegistriLetti[207] := ModBus.MB_Resp.Data[7];		(* Vedi tabella *)

				ModBus.MB_Query.Read_StartAddress := 209; (* richiedo lettura altri Parametri *)
				ModBus.MB_Query.Read_Quantity := 20;
				ModBus.MB_Start := TRUE;

				state := 55;
			END_IF
		END_IF

	55: (* Rispota Altri paramenti *)
		IF NOT ModBus.MB_Start  THEN

			IF ModBus.MB_MASTER.MB_Error<>0 THEN
				state := 300;
			ELSE
				MB_RegistriLetti[209] := ModBus.MB_Resp.Data[0];   	(* Vedi tabella *)
				MB_RegistriLetti[210] := ModBus.MB_Resp.Data[1];		(* Vedi tabella *)
				MB_RegistriLetti[211] := ModBus.MB_Resp.Data[2];		(* Vedi tabella *)
				MB_RegistriLetti[212] := ModBus.MB_Resp.Data[3];		(* Vedi tabella *)
				MB_RegistriLetti[213] := ModBus.MB_Resp.Data[4];		(* Vedi tabella *)
				MB_RegistriLetti[214] := ModBus.MB_Resp.Data[5];		(* Vedi tabella *)
				MB_RegistriLetti[215] := ModBus.MB_Resp.Data[6];		(* Vedi tabella *)
				MB_RegistriLetti[216] := ModBus.MB_Resp.Data[7];		(* Vedi tabella *)
				MB_RegistriLetti[217] := ModBus.MB_Resp.Data[8];		(* Vedi tabella *)
				MB_RegistriLetti[218] := ModBus.MB_Resp.Data[9];		(* Vedi tabella *)
				MB_RegistriLetti[219] := ModBus.MB_Resp.Data[10];		(* Vedi tabella *)
				MB_RegistriLetti[220] := ModBus.MB_Resp.Data[11];		(* Vedi tabella *)
				MB_RegistriLetti[221] := ModBus.MB_Resp.Data[12];		(* Vedi tabella *)
				MB_RegistriLetti[222] := ModBus.MB_Resp.Data[13];		(* Vedi tabella *)
				MB_RegistriLetti[223] := ModBus.MB_Resp.Data[14];		(* Vedi tabella *)
				MB_RegistriLetti[224] := ModBus.MB_Resp.Data[15];		(* Vedi tabella *)
				MB_RegistriLetti[225] := ModBus.MB_Resp.Data[16];		(* Vedi tabella *)
				MB_RegistriLetti[226] := ModBus.MB_Resp.Data[17];		(* Vedi tabella *)
				MB_RegistriLetti[227] := ModBus.MB_Resp.Data[18];		(* Vedi tabella *)
				MB_RegistriLetti[228] := ModBus.MB_Resp.Data[19];		(* Vedi tabella *)

				ModBus.MB_Query.Read_StartAddress := 229; (* richiedo lettura altri Parametri *)
				ModBus.MB_Query.Read_Quantity := 4;
				ModBus.MB_Start := TRUE;

				state := 60;
			END_IF
		END_IF

	60: (* Rispota Altri paramenti *)
		IF NOT ModBus.MB_Start  THEN

			IF ModBus.MB_MASTER.MB_Error<>0 THEN
				state := 300;
			ELSE
				MB_RegistriLetti[229] := ModBus.MB_Resp.Data[0];   	(* Vedi tabella *)
				MB_RegistriLetti[230] := ModBus.MB_Resp.Data[1];		(* Vedi tabella *)
				MB_RegistriLetti[231] := ModBus.MB_Resp.Data[2];		(* Vedi tabella *)
				MB_RegistriLetti[232] := ModBus.MB_Resp.Data[3];		(* Vedi tabella *)

				ModBus.MB_Query.Read_StartAddress := 235; (* richiedo lettura altri Parametri *)
				ModBus.MB_Query.Read_Quantity := 10;
				ModBus.MB_Start := TRUE;

				state := 65;
			END_IF
		END_IF


	65: (* Rispota Altri paramenti *)
		IF NOT ModBus.MB_Start  THEN

			IF ModBus.MB_MASTER.MB_Error<>0 THEN
				state := 300;
			ELSE
				MB_RegistriLetti[235] := ModBus.MB_Resp.Data[0];   	(* Vedi tabella *)
				MB_RegistriLetti[236] := ModBus.MB_Resp.Data[1];		(* Vedi tabella *)
				MB_RegistriLetti[237] := ModBus.MB_Resp.Data[2];		(* Vedi tabella *)
				MB_RegistriLetti[238] := ModBus.MB_Resp.Data[3];		(* Vedi tabella *)
				MB_RegistriLetti[239] := ModBus.MB_Resp.Data[4];		(* Vedi tabella *)
				MB_RegistriLetti[240] := ModBus.MB_Resp.Data[5];		(* Vedi tabella *)
				MB_RegistriLetti[241] := ModBus.MB_Resp.Data[6];		(* Vedi tabella *)
				MB_RegistriLetti[242] := ModBus.MB_Resp.Data[7];		(* Vedi tabella *)
				MB_RegistriLetti[243] := ModBus.MB_Resp.Data[8];		(* Vedi tabella *)
				MB_RegistriLetti[244] := ModBus.MB_Resp.Data[9];		(* Vedi tabella *)

				ModBus.MB_Query.Read_StartAddress := 268; (* richiedo lettura altri Parametri *)
				ModBus.MB_Query.Read_Quantity := 9;
				ModBus.MB_Start := TRUE;

				state := 70;
			END_IF
		END_IF

	70: (* Rispota Altri paramenti *)
		IF NOT ModBus.MB_Start  THEN

			IF ModBus.MB_MASTER.MB_Error<>0 THEN
				state := 300;
			ELSE
				MB_RegistriLetti[235] := ModBus.MB_Resp.Data[0];   	(* Vedi tabella *)
				MB_RegistriLetti[236] := ModBus.MB_Resp.Data[1];		(* Vedi tabella *)
				MB_RegistriLetti[237] := ModBus.MB_Resp.Data[2];		(* Vedi tabella *)
				MB_RegistriLetti[238] := ModBus.MB_Resp.Data[3];		(* Vedi tabella *)
				MB_RegistriLetti[239] := ModBus.MB_Resp.Data[4];		(* Vedi tabella *)
				MB_RegistriLetti[240] := ModBus.MB_Resp.Data[5];		(* Vedi tabella *)
				MB_RegistriLetti[241] := ModBus.MB_Resp.Data[6];		(* Vedi tabella *)
				MB_RegistriLetti[242] := ModBus.MB_Resp.Data[7];		(* Vedi tabella *)
				MB_RegistriLetti[243] := ModBus.MB_Resp.Data[8];		(* Vedi tabella *)
				MB_RegistriLetti[244] := ModBus.MB_Resp.Data[9];		(* Vedi tabella *)

				ModBus.MB_Query.Read_StartAddress := 268; (* richiedo lettura altri Parametri *)
				ModBus.MB_Query.Read_Quantity := 9;
				ModBus.MB_Start := TRUE;

				state := 75;
			END_IF
		END_IF


	75: (* Rispota Altri paramenti *)
		IF NOT ModBus.MB_Start  THEN

			IF ModBus.MB_MASTER.MB_Error<>0 THEN
				state := 300;
			ELSE
				MB_RegistriLetti[268] := ModBus.MB_Resp.Data[0];   	(* Vedi tabella *)
				MB_RegistriLetti[269] := ModBus.MB_Resp.Data[1];		(* Vedi tabella *)
				MB_RegistriLetti[270] := ModBus.MB_Resp.Data[2];		(* Vedi tabella *)
				MB_RegistriLetti[271] := ModBus.MB_Resp.Data[3];		(* Vedi tabella *)
				MB_RegistriLetti[272] := ModBus.MB_Resp.Data[4];		(* Vedi tabella *)
				MB_RegistriLetti[273] := ModBus.MB_Resp.Data[5];		(* Vedi tabella *)
				MB_RegistriLetti[274] := ModBus.MB_Resp.Data[6];		(* Vedi tabella *)
				MB_RegistriLetti[275] := ModBus.MB_Resp.Data[7];		(* Vedi tabella *)
				MB_RegistriLetti[276] := ModBus.MB_Resp.Data[8];		(* Vedi tabella *)

				ModBus.MB_Query.Read_StartAddress := 408; (* richiedo lettura altri Parametri *)
				ModBus.MB_Query.Read_Quantity := 6;
				ModBus.MB_Start := TRUE;

				state := 80;
			END_IF
		END_IF

	80: (* Rispota Altri paramenti *)
		IF NOT ModBus.MB_Start  THEN

			IF ModBus.MB_MASTER.MB_Error<>0 THEN
				state := 300;
			ELSE
				MB_RegistriLetti[408] := ModBus.MB_Resp.Data[0];   		(* Vedi tabella *)
				MB_RegistriLetti[409] := ModBus.MB_Resp.Data[1];		(* Vedi tabella *)
				MB_RegistriLetti[410] := ModBus.MB_Resp.Data[2];		(* Vedi tabella *)
				MB_RegistriLetti[411] := ModBus.MB_Resp.Data[3];		(* Vedi tabella *)
				MB_RegistriLetti[412] := ModBus.MB_Resp.Data[4];		(* Vedi tabella *)
				MB_RegistriLetti[413] := ModBus.MB_Resp.Data[5];		(* Vedi tabella *)

				ModBus.MB_Query.Read_StartAddress := 408; (* richiedo lettura altri Parametri *)
				ModBus.MB_Query.Read_Quantity := 6;
				ModBus.MB_Start := TRUE;

				state := 100;
			END_IF
		END_IF






	100: (* Rispota Altri paramenti COIL *)
		IF NOT ModBus.MB_Start  THEN

			IF ModBus.MB_MASTER.MB_Error<>0 THEN
				state := 300;
			ELSE
				Modbus.MB_Query.SlaveAddress := Address;
				Modbus.MB_Query.FunctionCode := 1;
				ModBus.MB_Query.Read_StartAddress := 0;	(* richiedo lettura altri Parametri *)
				ModBus.MB_Query.Read_Quantity := 60;
				ModBus.MB_Start := TRUE;

				state:=105;
			END_IF
		END_IF
	105: (* Rispota Altri paramenti *)

		IF NOT ModBus.MB_Start  THEN

			IF ModBus.MB_MASTER.MB_Error<>0 THEN
				state := 300;
			ELSE

				MB_BitStato[0]:=ModBus.MB_MASTER.ReceiveBuffer.Data[3].0; (*Vedi Tabella *)
				MB_BitStato[1]:=ModBus.MB_MASTER.ReceiveBuffer.Data[3].1; (*Vedi Tabella *)
				MB_BitStato[2]:=ModBus.MB_MASTER.ReceiveBuffer.Data[3].2; (*Vedi Tabella *)
				MB_BitStato[3]:=ModBus.MB_MASTER.ReceiveBuffer.Data[3].3; (*Vedi Tabella *)
				MB_BitStato[4]:=ModBus.MB_MASTER.ReceiveBuffer.Data[3].4; (*Vedi Tabella *)
				MB_BitStato[5]:=ModBus.MB_MASTER.ReceiveBuffer.Data[3].5; (*Vedi Tabella *)
				MB_BitStato[6]:=ModBus.MB_MASTER.ReceiveBuffer.Data[3].6; (*Vedi Tabella *)
				MB_BitStato[7]:=ModBus.MB_MASTER.ReceiveBuffer.Data[3].7; (*Vedi Tabella *)
				MB_BitStato[8]:=ModBus.MB_MASTER.ReceiveBuffer.Data[4].0; (*Vedi Tabella *)
				MB_BitStato[9]:=ModBus.MB_MASTER.ReceiveBuffer.Data[4].1; (*Vedi Tabella *)
				MB_BitStato[10]:=ModBus.MB_MASTER.ReceiveBuffer.Data[4].2; (*Vedi Tabella *)
				MB_BitStato[11]:=ModBus.MB_MASTER.ReceiveBuffer.Data[4].3; (*Vedi Tabella *)
				MB_BitStato[12]:=ModBus.MB_MASTER.ReceiveBuffer.Data[4].4; (*Vedi Tabella *)
				MB_BitStato[13]:=ModBus.MB_MASTER.ReceiveBuffer.Data[4].5; (*Vedi Tabella *)
				MB_BitStato[14]:=ModBus.MB_MASTER.ReceiveBuffer.Data[4].6; (*Vedi Tabella *)
				MB_BitStato[15]:=ModBus.MB_MASTER.ReceiveBuffer.Data[4].7; (*Vedi Tabella *)
				MB_BitStato[16]:=ModBus.MB_MASTER.ReceiveBuffer.Data[5].0; (*Vedi Tabella *)
				MB_BitStato[17]:=ModBus.MB_MASTER.ReceiveBuffer.Data[5].1; (*Vedi Tabella *)
				MB_BitStato[18]:=ModBus.MB_MASTER.ReceiveBuffer.Data[5].2; (*Vedi Tabella *)
				MB_BitStato[19]:=ModBus.MB_MASTER.ReceiveBuffer.Data[5].3; (*Vedi Tabella *)
				MB_BitStato[20]:=ModBus.MB_MASTER.ReceiveBuffer.Data[5].4; (*Vedi Tabella *)
				MB_BitStato[21]:=ModBus.MB_MASTER.ReceiveBuffer.Data[5].5; (*Vedi Tabella *)
				MB_BitStato[22]:=ModBus.MB_MASTER.ReceiveBuffer.Data[5].6; (*Vedi Tabella *)
				MB_BitStato[23]:=ModBus.MB_MASTER.ReceiveBuffer.Data[5].7; (*Vedi Tabella *)
				MB_BitStato[24]:=ModBus.MB_MASTER.ReceiveBuffer.Data[6].0; (*Vedi Tabella *)
				MB_BitStato[25]:=ModBus.MB_MASTER.ReceiveBuffer.Data[6].1; (*Vedi Tabella *)
				MB_BitStato[26]:=ModBus.MB_MASTER.ReceiveBuffer.Data[6].2; (*Vedi Tabella *)
				MB_BitStato[27]:=ModBus.MB_MASTER.ReceiveBuffer.Data[6].3; (*Vedi Tabella *)
				MB_BitStato[28]:=ModBus.MB_MASTER.ReceiveBuffer.Data[6].4; (*Vedi Tabella *)
				MB_BitStato[29]:=ModBus.MB_MASTER.ReceiveBuffer.Data[6].5; (*Vedi Tabella *)
				MB_BitStato[30]:=ModBus.MB_MASTER.ReceiveBuffer.Data[6].6; (*Vedi Tabella *)
				MB_BitStato[31]:=ModBus.MB_MASTER.ReceiveBuffer.Data[6].7; (*Vedi Tabella *)
				MB_BitStato[32]:=ModBus.MB_MASTER.ReceiveBuffer.Data[7].0; (*Vedi Tabella *)
				MB_BitStato[33]:=ModBus.MB_MASTER.ReceiveBuffer.Data[7].1; (*Vedi Tabella *)
				MB_BitStato[34]:=ModBus.MB_MASTER.ReceiveBuffer.Data[7].2; (*Vedi Tabella *)
				MB_BitStato[35]:=ModBus.MB_MASTER.ReceiveBuffer.Data[7].3; (*Vedi Tabella *)
				MB_BitStato[36]:=ModBus.MB_MASTER.ReceiveBuffer.Data[7].4; (*Vedi Tabella *)
				MB_BitStato[37]:=ModBus.MB_MASTER.ReceiveBuffer.Data[7].5; (*Vedi Tabella *)
				MB_BitStato[38]:=ModBus.MB_MASTER.ReceiveBuffer.Data[7].6; (*Vedi Tabella *)
				MB_BitStato[39]:=ModBus.MB_MASTER.ReceiveBuffer.Data[7].7; (*Vedi Tabella *)
				MB_BitStato[40]:=ModBus.MB_MASTER.ReceiveBuffer.Data[8].0; (*Vedi Tabella *)
				MB_BitStato[41]:=ModBus.MB_MASTER.ReceiveBuffer.Data[8].1; (*Vedi Tabella *)
				MB_BitStato[42]:=ModBus.MB_MASTER.ReceiveBuffer.Data[8].2; (*Vedi Tabella *)
				MB_BitStato[43]:=ModBus.MB_MASTER.ReceiveBuffer.Data[8].3; (*Vedi Tabella *)
				MB_BitStato[44]:=ModBus.MB_MASTER.ReceiveBuffer.Data[8].4; (*Vedi Tabella *)
				MB_BitStato[45]:=ModBus.MB_MASTER.ReceiveBuffer.Data[8].5; (*Vedi Tabella *)
				MB_BitStato[46]:=ModBus.MB_MASTER.ReceiveBuffer.Data[8].6; (*Vedi Tabella *)
				MB_BitStato[47]:=ModBus.MB_MASTER.ReceiveBuffer.Data[8].7; (*Vedi Tabella *)
				MB_BitStato[48]:=ModBus.MB_MASTER.ReceiveBuffer.Data[9].0; (*Vedi Tabella *)
				MB_BitStato[49]:=ModBus.MB_MASTER.ReceiveBuffer.Data[9].1; (*Vedi Tabella *)
				MB_BitStato[50]:=ModBus.MB_MASTER.ReceiveBuffer.Data[9].2; (*Vedi Tabella *)
				MB_BitStato[51]:=ModBus.MB_MASTER.ReceiveBuffer.Data[9].3; (*Vedi Tabella *)
				MB_BitStato[52]:=ModBus.MB_MASTER.ReceiveBuffer.Data[9].4; (*Vedi Tabella *)
				MB_BitStato[53]:=ModBus.MB_MASTER.ReceiveBuffer.Data[9].5; (*Vedi Tabella *)
				MB_BitStato[54]:=ModBus.MB_MASTER.ReceiveBuffer.Data[9].6; (*Vedi Tabella *)
				MB_BitStato[55]:=ModBus.MB_MASTER.ReceiveBuffer.Data[9].7; (*Vedi Tabella *)
				MB_BitStato[56]:=ModBus.MB_MASTER.ReceiveBuffer.Data[10].0; (*Vedi Tabella *)
				MB_BitStato[57]:=ModBus.MB_MASTER.ReceiveBuffer.Data[10].1; (*Vedi Tabella *)
				MB_BitStato[58]:=ModBus.MB_MASTER.ReceiveBuffer.Data[10].2; (*Vedi Tabella *)
				MB_BitStato[59]:=ModBus.MB_MASTER.ReceiveBuffer.Data[10].3; (*Vedi Tabella *)
				MB_BitStato[60]:=ModBus.MB_MASTER.ReceiveBuffer.Data[10].4; (*Vedi Tabella *)
				MB_BitStato[61]:=ModBus.MB_MASTER.ReceiveBuffer.Data[10].5; (*Vedi Tabella *)
				MB_BitStato[62]:=ModBus.MB_MASTER.ReceiveBuffer.Data[10].6; (*Vedi Tabella *)
				MB_BitStato[63]:=ModBus.MB_MASTER.ReceiveBuffer.Data[10].7; (*Vedi Tabella *)


				state:=110;

			END_IF
		END_IF


	110: (* Rispota Altri paramenti *)
		IF NOT ModBus.MB_Start  THEN

			IF ModBus.MB_MASTER.MB_Error<>0 THEN
				state := 300;
			ELSE
				Modbus.MB_Query.SlaveAddress := Address;
				Modbus.MB_Query.FunctionCode := 1;
				ModBus.MB_Query.Read_StartAddress := 100;
				ModBus.MB_Query.Read_Quantity := 100;
				ModBus.MB_Start := TRUE;

				state:=115;
			END_IF
		END_IF
	115: (* Rispota Altri paramenti *)

		IF NOT ModBus.MB_Start  THEN

			IF ModBus.MB_MASTER.MB_Error<>0 THEN
				state := 300;
			ELSE

				MB_BitStato[100]:=ModBus.MB_MASTER.ReceiveBuffer.Data[3].0; (*Vedi Tabella *)
				MB_BitStato[101]:=ModBus.MB_MASTER.ReceiveBuffer.Data[3].1; (*Vedi Tabella *)
				MB_BitStato[102]:=ModBus.MB_MASTER.ReceiveBuffer.Data[3].2; (*Vedi Tabella *)
				MB_BitStato[103]:=ModBus.MB_MASTER.ReceiveBuffer.Data[3].3; (*Vedi Tabella *)
				MB_BitStato[104]:=ModBus.MB_MASTER.ReceiveBuffer.Data[3].4; (*Vedi Tabella *)
				MB_BitStato[105]:=ModBus.MB_MASTER.ReceiveBuffer.Data[3].5; (*Vedi Tabella *)
				MB_BitStato[106]:=ModBus.MB_MASTER.ReceiveBuffer.Data[3].6; (*Vedi Tabella *)
				MB_BitStato[107]:=ModBus.MB_MASTER.ReceiveBuffer.Data[3].7; (*Vedi Tabella *)
				MB_BitStato[108]:=ModBus.MB_MASTER.ReceiveBuffer.Data[4].0; (*Vedi Tabella *)
				MB_BitStato[109]:=ModBus.MB_MASTER.ReceiveBuffer.Data[4].1; (*Vedi Tabella *)
				MB_BitStato[110]:=ModBus.MB_MASTER.ReceiveBuffer.Data[4].2; (*Vedi Tabella *)
				MB_BitStato[111]:=ModBus.MB_MASTER.ReceiveBuffer.Data[4].3; (*Vedi Tabella *)
				MB_BitStato[112]:=ModBus.MB_MASTER.ReceiveBuffer.Data[4].4; (*Vedi Tabella *)
				MB_BitStato[113]:=ModBus.MB_MASTER.ReceiveBuffer.Data[4].5; (*Vedi Tabella *)
				MB_BitStato[114]:=ModBus.MB_MASTER.ReceiveBuffer.Data[4].6; (*Vedi Tabella *)
				MB_BitStato[115]:=ModBus.MB_MASTER.ReceiveBuffer.Data[4].7; (*Vedi Tabella *)
				MB_BitStato[116]:=ModBus.MB_MASTER.ReceiveBuffer.Data[5].0; (*Vedi Tabella *)
				MB_BitStato[117]:=ModBus.MB_MASTER.ReceiveBuffer.Data[5].1; (*Vedi Tabella *)
				MB_BitStato[118]:=ModBus.MB_MASTER.ReceiveBuffer.Data[5].2; (*Vedi Tabella *)
				MB_BitStato[119]:=ModBus.MB_MASTER.ReceiveBuffer.Data[5].3; (*Vedi Tabella *)
				MB_BitStato[120]:=ModBus.MB_MASTER.ReceiveBuffer.Data[5].4; (*Vedi Tabella *)
				MB_BitStato[121]:=ModBus.MB_MASTER.ReceiveBuffer.Data[5].5; (*Vedi Tabella *)
				MB_BitStato[122]:=ModBus.MB_MASTER.ReceiveBuffer.Data[5].6; (*Vedi Tabella *)
				MB_BitStato[123]:=ModBus.MB_MASTER.ReceiveBuffer.Data[5].7; (*Vedi Tabella *)
				MB_BitStato[124]:=ModBus.MB_MASTER.ReceiveBuffer.Data[6].0; (*Vedi Tabella *)
				MB_BitStato[125]:=ModBus.MB_MASTER.ReceiveBuffer.Data[6].1; (*Vedi Tabella *)
				MB_BitStato[126]:=ModBus.MB_MASTER.ReceiveBuffer.Data[6].2; (*Vedi Tabella *)
				MB_BitStato[127]:=ModBus.MB_MASTER.ReceiveBuffer.Data[6].3; (*Vedi Tabella *)
				MB_BitStato[128]:=ModBus.MB_MASTER.ReceiveBuffer.Data[6].4; (*Vedi Tabella *)
				MB_BitStato[129]:=ModBus.MB_MASTER.ReceiveBuffer.Data[6].5; (*Vedi Tabella *)
				MB_BitStato[130]:=ModBus.MB_MASTER.ReceiveBuffer.Data[6].6; (*Vedi Tabella *)
				MB_BitStato[131]:=ModBus.MB_MASTER.ReceiveBuffer.Data[6].7; (*Vedi Tabella *)
				MB_BitStato[132]:=ModBus.MB_MASTER.ReceiveBuffer.Data[7].0; (*Vedi Tabella *)
				MB_BitStato[133]:=ModBus.MB_MASTER.ReceiveBuffer.Data[7].1; (*Vedi Tabella *)
				MB_BitStato[134]:=ModBus.MB_MASTER.ReceiveBuffer.Data[7].2; (*Vedi Tabella *)
				MB_BitStato[135]:=ModBus.MB_MASTER.ReceiveBuffer.Data[7].3; (*Vedi Tabella *)
				MB_BitStato[136]:=ModBus.MB_MASTER.ReceiveBuffer.Data[7].4; (*Vedi Tabella *)
				MB_BitStato[137]:=ModBus.MB_MASTER.ReceiveBuffer.Data[7].5; (*Vedi Tabella *)
				MB_BitStato[138]:=ModBus.MB_MASTER.ReceiveBuffer.Data[7].6; (*Vedi Tabella *)
				MB_BitStato[139]:=ModBus.MB_MASTER.ReceiveBuffer.Data[7].7; (*Vedi Tabella *)
				MB_BitStato[140]:=ModBus.MB_MASTER.ReceiveBuffer.Data[8].0; (*Vedi Tabella *)
				MB_BitStato[141]:=ModBus.MB_MASTER.ReceiveBuffer.Data[8].1; (*Vedi Tabella *)
				MB_BitStato[142]:=ModBus.MB_MASTER.ReceiveBuffer.Data[8].2; (*Vedi Tabella *)
				MB_BitStato[143]:=ModBus.MB_MASTER.ReceiveBuffer.Data[8].3; (*Vedi Tabella *)
				MB_BitStato[144]:=ModBus.MB_MASTER.ReceiveBuffer.Data[8].4; (*Vedi Tabella *)
				MB_BitStato[145]:=ModBus.MB_MASTER.ReceiveBuffer.Data[8].5; (*Vedi Tabella *)
				MB_BitStato[146]:=ModBus.MB_MASTER.ReceiveBuffer.Data[8].6; (*Vedi Tabella *)
				MB_BitStato[147]:=ModBus.MB_MASTER.ReceiveBuffer.Data[8].7; (*Vedi Tabella *)
				MB_BitStato[148]:=ModBus.MB_MASTER.ReceiveBuffer.Data[9].0; (*Vedi Tabella *)
				MB_BitStato[149]:=ModBus.MB_MASTER.ReceiveBuffer.Data[9].1; (*Vedi Tabella *)
				MB_BitStato[150]:=ModBus.MB_MASTER.ReceiveBuffer.Data[9].2; (*Vedi Tabella *)
				MB_BitStato[151]:=ModBus.MB_MASTER.ReceiveBuffer.Data[9].3; (*Vedi Tabella *)
				MB_BitStato[152]:=ModBus.MB_MASTER.ReceiveBuffer.Data[9].4; (*Vedi Tabella *)
				MB_BitStato[153]:=ModBus.MB_MASTER.ReceiveBuffer.Data[9].5; (*Vedi Tabella *)
				MB_BitStato[154]:=ModBus.MB_MASTER.ReceiveBuffer.Data[9].6; (*Vedi Tabella *)
				MB_BitStato[155]:=ModBus.MB_MASTER.ReceiveBuffer.Data[9].7; (*Vedi Tabella *)
				MB_BitStato[156]:=ModBus.MB_MASTER.ReceiveBuffer.Data[10].0; (*Vedi Tabella *)
				MB_BitStato[157]:=ModBus.MB_MASTER.ReceiveBuffer.Data[10].1; (*Vedi Tabella *)
				MB_BitStato[158]:=ModBus.MB_MASTER.ReceiveBuffer.Data[10].2; (*Vedi Tabella *)
				MB_BitStato[159]:=ModBus.MB_MASTER.ReceiveBuffer.Data[10].3; (*Vedi Tabella *)
				MB_BitStato[160]:=ModBus.MB_MASTER.ReceiveBuffer.Data[10].4; (*Vedi Tabella *)
				MB_BitStato[161]:=ModBus.MB_MASTER.ReceiveBuffer.Data[10].5; (*Vedi Tabella *)
				MB_BitStato[162]:=ModBus.MB_MASTER.ReceiveBuffer.Data[10].6; (*Vedi Tabella *)
				MB_BitStato[163]:=ModBus.MB_MASTER.ReceiveBuffer.Data[10].7; (*Vedi Tabella *)
				MB_BitStato[164]:=ModBus.MB_MASTER.ReceiveBuffer.Data[11].0; (*Vedi Tabella *)
				MB_BitStato[165]:=ModBus.MB_MASTER.ReceiveBuffer.Data[11].1; (*Vedi Tabella *)
				MB_BitStato[166]:=ModBus.MB_MASTER.ReceiveBuffer.Data[11].2; (*Vedi Tabella *)
				MB_BitStato[167]:=ModBus.MB_MASTER.ReceiveBuffer.Data[11].3; (*Vedi Tabella *)
				MB_BitStato[168]:=ModBus.MB_MASTER.ReceiveBuffer.Data[11].4; (*Vedi Tabella *)
				MB_BitStato[169]:=ModBus.MB_MASTER.ReceiveBuffer.Data[11].5; (*Vedi Tabella *)
				MB_BitStato[170]:=ModBus.MB_MASTER.ReceiveBuffer.Data[11].6; (*Vedi Tabella *)
				MB_BitStato[171]:=ModBus.MB_MASTER.ReceiveBuffer.Data[11].7; (*Vedi Tabella *)
				MB_BitStato[172]:=ModBus.MB_MASTER.ReceiveBuffer.Data[12].0; (*Vedi Tabella *)
				MB_BitStato[173]:=ModBus.MB_MASTER.ReceiveBuffer.Data[12].1; (*Vedi Tabella *)
				MB_BitStato[174]:=ModBus.MB_MASTER.ReceiveBuffer.Data[12].2; (*Vedi Tabella *)
				MB_BitStato[175]:=ModBus.MB_MASTER.ReceiveBuffer.Data[12].3; (*Vedi Tabella *)
				MB_BitStato[176]:=ModBus.MB_MASTER.ReceiveBuffer.Data[12].4; (*Vedi Tabella *)
				MB_BitStato[177]:=ModBus.MB_MASTER.ReceiveBuffer.Data[12].5; (*Vedi Tabella *)
				MB_BitStato[178]:=ModBus.MB_MASTER.ReceiveBuffer.Data[12].6; (*Vedi Tabella *)
				MB_BitStato[179]:=ModBus.MB_MASTER.ReceiveBuffer.Data[12].7; (*Vedi Tabella *)
				MB_BitStato[180]:=ModBus.MB_MASTER.ReceiveBuffer.Data[13].0; (*Vedi Tabella *)
				MB_BitStato[181]:=ModBus.MB_MASTER.ReceiveBuffer.Data[13].1; (*Vedi Tabella *)
				MB_BitStato[182]:=ModBus.MB_MASTER.ReceiveBuffer.Data[13].2; (*Vedi Tabella *)
				MB_BitStato[183]:=ModBus.MB_MASTER.ReceiveBuffer.Data[13].3; (*Vedi Tabella *)
				MB_BitStato[184]:=ModBus.MB_MASTER.ReceiveBuffer.Data[13].4; (*Vedi Tabella *)
				MB_BitStato[185]:=ModBus.MB_MASTER.ReceiveBuffer.Data[13].5; (*Vedi Tabella *)
				MB_BitStato[186]:=ModBus.MB_MASTER.ReceiveBuffer.Data[13].6; (*Vedi Tabella *)
				MB_BitStato[187]:=ModBus.MB_MASTER.ReceiveBuffer.Data[13].7; (*Vedi Tabella *)
				MB_BitStato[188]:=ModBus.MB_MASTER.ReceiveBuffer.Data[13].0; (*Vedi Tabella *)
				MB_BitStato[189]:=ModBus.MB_MASTER.ReceiveBuffer.Data[13].1; (*Vedi Tabella *)
				MB_BitStato[190]:=ModBus.MB_MASTER.ReceiveBuffer.Data[13].2; (*Vedi Tabella *)
				MB_BitStato[191]:=ModBus.MB_MASTER.ReceiveBuffer.Data[13].3; (*Vedi Tabella *)
				MB_BitStato[192]:=ModBus.MB_MASTER.ReceiveBuffer.Data[13].4; (*Vedi Tabella *)
				MB_BitStato[193]:=ModBus.MB_MASTER.ReceiveBuffer.Data[13].5; (*Vedi Tabella *)
				MB_BitStato[194]:=ModBus.MB_MASTER.ReceiveBuffer.Data[13].6; (*Vedi Tabella *)
				MB_BitStato[195]:=ModBus.MB_MASTER.ReceiveBuffer.Data[13].7; (*Vedi Tabella *)
				MB_BitStato[196]:=ModBus.MB_MASTER.ReceiveBuffer.Data[14].0; (*Vedi Tabella *)
				MB_BitStato[197]:=ModBus.MB_MASTER.ReceiveBuffer.Data[14].1; (*Vedi Tabella *)
				MB_BitStato[198]:=ModBus.MB_MASTER.ReceiveBuffer.Data[14].2; (*Vedi Tabella *)
				MB_BitStato[199]:=ModBus.MB_MASTER.ReceiveBuffer.Data[14].3; (*Vedi Tabella *)


				state:=290;

			END_IF
		END_IF




		290:    (* Scrittura BOOL - COIL o WORD *)
		IF NOT ModBus.MB_Start THEN
			IF ModBus.MB_MASTER.MB_Error<>0 THEN (*OR ModBus.MB_MASTER.MB_Error<>0 THEN*)
				state := 300;
			ELSE
				IF ScriviDato THEN
					IF ScriviCoil THEN
						Modbus.MB_Query.FunctionCode := 5;
					ELSE
						Modbus.MB_Query.FunctionCode := 6;
					END_IF
					Modbus.MB_Query.SlaveAddress := Address;
					ModBus.MB_Query.Write_StartAddress := IndirizzoDaScrivere;
					ModBus.MB_Query.Write_Quantity :=1;
					ModBus.MB_Query.Write_Data[0] := DatoDaScrivere;
					ModBus.MB_Start := TRUE;
						IF ScriviCoil THEN
							IF 	MB_BitStato[IndirizzoDaScrivere]=WORD_TO_BOOL(DatoDaScrivere-1) THEN
								ScriviDato:=FALSE;
							END_IF
						ELSE
							IF 	MB_RegistriLetti[IndirizzoDaScrivere]=DatoDaScrivere THEN
								ScriviDato:=FALSE;
							END_IF
						END_IF
					state := 295;
				ELSE
					state := 295;
				END_IF
			END_IF
		END_IF




		295:
		IF NOT ModBus.MB_Start THEN
			IF ModBus.MB_MASTER.MB_Error<>0 THEN (*OR ModBus.MB_MASTER.MB_Error<>0 THEN*)
				state := 300;
			ELSE
				IF fModbusAlr THEN fModbusAlr := FALSE; END_IF
				NodoDaInterrogareChiller:=Address+1;
				InibiscoModbusChiller:=FALSE;
				retryErr := 0;
				retry := 0;
				state := 0;
					IF fModbusAlr=FALSE AND ErroreComuModBus=TRUE THEN
						LogEv(EL_Log,EO_CHI,ID,62,'ComunicazioneModBus_OK');
						ErroreComuModBus := FALSE;
				(*	WarningCtr := SEL(WarningCtr=0, WarningCtr-1, 0); *)
					END_IF


			END_IF
		END_IF



	(**** CHECK MODBUS ERROR ****)
	300: 	(* Release MODBUS *)
			InibiscoModbusChiller:=FALSE;
			(* Retries *)
			retry:=retry+1;
			IF retry>3 THEN
				retry:=0;

				(* Verify if slave is dead *)
				IF retryErr < retryErrMaX THEN
					retryErr := retryErr + 1;
				ELSE
					fModbusAlr := TRUE;
					(* Verify ModBus error	*)

					IF fModbusAlr AND ErroreComuModBus=FALSE THEN
						LogEv(EL_Alarm,EO_CHI,ID,61,CONCAT('ErroreModbus_',INT_TO_STRING(ModBus.MB_MASTER.MB_Error)));
						ErroreComuModBus := TRUE;
					END_IF
				END_IF

				END_IF
			Refresh_Now := FALSE;
			NodoDaInterrogareChiller:=Address+1;
			state:=0;
END_CASE




(* Controllo Time Out Ciclo ModBus *)

TimeOutModBus(In:=state<>0,PT:=t#30s);
IF TimeOutModBus.Q THEN
	State:=0;
	Refresh_Now:=TRUE;  (* Rilancio la lettura del nodo *)
	IF MODBUS.MB_Lock=TRUE THEN MODBUS.MB_Lock:=FALSE;END_IF
	IF InibiscoModbusChiller=TRUE THEN InibiscoModbusChiller:=FALSE;END_IF
END_IF
END_ACTION

(* POU Utils Functions/TONOF, ST *)
FUNCTION_BLOCK TONOF
VAR_INPUT
	IN		: BOOL;
	PT_ON	: TIME; (* time to pass, before OUT is set *)
	PT_OF	: TIME; (* time to pass, before OUT is reset *)
END_VAR
VAR_OUTPUT
	OUT		: BOOL;
END_VAR
VAR
	timer	: TON;
END_VAR
IF IN<>OUT THEN
	timer(IN:=TRUE,PT:=SEL(IN,PT_OF,PT_ON));
	IF timer.Q THEN OUT:=IN; END_IF
ELSE
	timer(IN:=FALSE);
END_IF
END_FUNCTION_BLOCK

(* POU Plant_Objects/obj_MODBUS_TRENDCOIN_01, ST *)
FUNCTION_BLOCK obj_MODBUS_TRENDCOIN_01
VAR CONSTANT

	TimeOutModBus: TON;


END_VAR
VAR_INPUT
	ID			:	BYTE;
	Address		:	BYTE;
	(* Modbus *)
	Refresh_Now	:	BOOL;			(* Richiesta di lettura stato macchina Immediata  *)
	retryErrMax	:	BYTE := 2;

	IndirizzoDaScrivere: WORD;
	DatoDaScrivere: INT;
	ScriviDato: BOOL;
	ScriviCoil: BOOL;

(* Variabili da scrivere nel parametri Trend *)

	EnScrittura		:ARRAY [0..15] OF	FLT_EVENT;


	Abilita_UTA01:BOOL;
	Abilita_UTA02:BOOL;
	Abilita_UTA03:BOOL;
	Abilita_UTA04:BOOL;
	Abilita_UTA05:BOOL;
	Abilita_UTA06:BOOL;
	Abilita_UTA07:BOOL;
	Abilita_UTA08:BOOL;
	Abilita_UTA09:BOOL;
	Abilita_UTA10:BOOL;
	Abilita_UTA12:BOOL;
	Abilita_UTA13:BOOL;



END_VAR
VAR_IN_OUT
	ModBus		:obj_MODBUS;

END_VAR
VAR_OUTPUT
	Status_Log	:	WORD;
	Status_Vis	:	DWORD;
END_VAR
VAR

	state		:	INT;
	retry		:	BYTE;
	retryErr	:	BYTE;
	ReadTmr		:	TON := (PT:=T#5s);
	fModbusAlr:BOOL;

(*	retry_write	:	BYTE;
	fWriteStatus:	BOOL;
	fWriteMode	:	BOOL;
	fWriteReset	:	BOOL; *)

	x: INT;

	VerificaFuctionCode: INT;
	VerificaNodoLetto: INT;
	ErroreComuModBus: BOOL;
	IndiceErrore: BYTE;

	MB_BitStato: ARRAY [0..450] OF BOOL;
	MB_RegistriLetti: ARRAY [0..450] OF INT;
	MB_RegistriHoldingLetti: ARRAY [0..170] OF INT;
	MB_BitStatoCoil: ARRAY [0..100] OF BOOL;




	AddressRead: BYTE;
	index: BYTE;
	indexErr: BYTE;


	Read_StartAddress: INT;
	Read_Quantity: BYTE;
	IndiceMBLettura: INT;
	IndiceMBLetto: INT;



	test_Address: INT;
	Test_ScriviCoil: BOOL;
	test_Write: WORD;
	ScriviMB: BOOL;


	ScriviRUN_UTA01:BOOL;
	ScriviRUN_UTA02:BOOL;
	ScriviRUN_UTA03:BOOL;
	ScriviRUN_UTA04:BOOL;
	ScriviRUN_UTA05:BOOL;
	ScriviRUN_UTA06:BOOL;
	ScriviRUN_UTA07:BOOL;
	ScriviRUN_UTA08:BOOL;
	ScriviRUN_UTA09:BOOL;
	ScriviRUN_UTA10:BOOL;
	ScriviRUN_UTA12:BOOL;
	ScriviRUN_UTA13:BOOL;








	AddressDaScrivere: INT;


	temp :STRING(255);
	tempRaw		: ARRAY [0..MAX_SEND_TCP_CLIENT] OF BYTE;
	tempRawLen :DINT;
	longString:STRING(800);







END_VAR
	EnScrittura[1](IN:=Abilita_UTA01);
	ScriviRUN_UTA01:=EnScrittura[1].EVH;
	ScriviRUN_UTA01:=EnScrittura[1].EVL;

	EnScrittura[2](IN:=Abilita_UTA02);
	ScriviRUN_UTA02:=EnScrittura[2].EVH;
	ScriviRUN_UTA02:=EnScrittura[2].EVL;

	EnScrittura[3](IN:=Abilita_UTA03);
	ScriviRUN_UTA03:=EnScrittura[3].EVH;
	ScriviRUN_UTA03:=EnScrittura[3].EVL;

	EnScrittura[4](IN:=Abilita_UTA04);
	ScriviRUN_UTA04:=EnScrittura[4].EVH;
	ScriviRUN_UTA04:=EnScrittura[4].EVL;

	EnScrittura[4](IN:=Abilita_UTA04);
	ScriviRUN_UTA04:=EnScrittura[4].EVH;
	ScriviRUN_UTA04:=EnScrittura[4].EVL;

	EnScrittura[5](IN:=Abilita_UTA05);
	ScriviRUN_UTA05:=EnScrittura[5].EVH;
	ScriviRUN_UTA05:=EnScrittura[5].EVL;

	EnScrittura[6](IN:=Abilita_UTA06);
	ScriviRUN_UTA06:=EnScrittura[6].EVH;
	ScriviRUN_UTA06:=EnScrittura[6].EVL;

	EnScrittura[7](IN:=Abilita_UTA07);
	ScriviRUN_UTA07:=EnScrittura[7].EVH;
	ScriviRUN_UTA07:=EnScrittura[7].EVL;

	EnScrittura[8](IN:=Abilita_UTA08);
	ScriviRUN_UTA08:=EnScrittura[8].EVH;
	ScriviRUN_UTA08:=EnScrittura[8].EVL;

	EnScrittura[9](IN:=Abilita_UTA09);
	ScriviRUN_UTA09:=EnScrittura[9].EVH;
	ScriviRUN_UTA09:=EnScrittura[9].EVL;

	EnScrittura[10](IN:=Abilita_UTA10);
	ScriviRUN_UTA10:=EnScrittura[10].EVH;
	ScriviRUN_UTA10:=EnScrittura[10].EVL;

(*	EnScrittura[11](IN:=Abilita_UTA11);
	ScriviRUN_UTA11:=EnScrittura[11].EVH;
	ScriviRUN_UTA11:=EnScrittura[11].EVL; *)

	EnScrittura[12](IN:=Abilita_UTA12);
	ScriviRUN_UTA12:=EnScrittura[12].EVH;
	ScriviRUN_UTA12:=EnScrittura[12].EVL;

	EnScrittura[13](IN:=Abilita_UTA13);
	ScriviRUN_UTA13:=EnScrittura[13].EVH;
	ScriviRUN_UTA13:=EnScrittura[13].EVL;






(* Call ModBus state machine *)
Stm();

(* Check alarm	*)




(* Seganalzione stato Frigorifero  *)
IF ErroreComuModBus THEN
		Status_Log:=2; Status_Vis:=16#2020F0;
(*	ELSIF Warning OR Warning2 THEN
		Status_Log:=1; Status_Vis:=16#20F0F0; *)
    ELSE
		Status_Log:=0;
		Status_Vis:=16#006000;
END_IF
END_FUNCTION_BLOCK
ACTION AddLogData:
Logger.s1:=INSERT('&POOL=',BYTE_TO_STRING(ID),5);
IF ID<10 THEN Logger.s1:=INSERT(Logger.s1,'0',5); END_IF


(* inizializzo stringa da loggare **)
FOR tempRawLen:=0 TO MAX_SEND_TCP_CLIENT DO
                tempRaw[tempRawLen]:=0;
END_FOR

tempRawLen:=0;


